	VAR robtarget Openhole_2763 := [[394.33, -31.54, 174.56], [-0.132881, 0.694509, 0.676037, 0.207303], [0,0,0,0], [9E9, 9E9, 9E9, 9E9, 9E9, 9E9]];
	VAR robtarget Openhole_2764 := [[389.32, -31.54, 173.95], [-0.146442, 0.691776, 0.672345, 0.218979], [0,0,0,0], [9E9, 9E9, 9E9, 9E9, 9E9, 9E9]];
	VAR robtarget Openhole_2765 := [[362.32, -31.54, 174.04], [-0.183051, 0.683002, 0.683002, 0.183051], [0,0,0,0], [9E9, 9E9, 9E9, 9E9, 9E9, 9E9]];
	VAR robtarget Openhole_2766 := [[362.32, -32.55, 173.46], [-0.183051, 0.683002, 0.683002, 0.183051], [0,0,0,0], [9E9, 9E9, 9E9, 9E9, 9E9, 9E9]];
	VAR robtarget Openhole_2767 := [[389.32, -32.55, 173.37], [-0.143577, 0.692377, 0.671432, 0.221765], [0,0,0,0], [9E9, 9E9, 9E9, 9E9, 9E9, 9E9]];
	VAR robtarget Openhole_2768 := [[394.32, -32.55, 174.02], [-0.129957, 0.695062, 0.675151, 0.210168], [0,0,0,0], [9E9, 9E9, 9E9, 9E9, 9E9, 9E9]];
	VAR robtarget Openhole_2769 := [[395.25, -32.64, 174.1], [-0.127122, 0.695586, 0.675755, 0.20822], [0,0,0,0], [9E9, 9E9, 9E9, 9E9, 9E9, 9E9]];
	VAR robtarget Openhole_2770 := [[405.09, -34.29, 174.68], [-0.093512, 0.700896, 0.681563, 0.188339], [0,0,0,0], [9E9, 9E9, 9E9, 9E9, 9E9, 9E9]];
	VAR robtarget Openhole_2771 := [[411.51, -35.11, 175.33], [-0.071164, 0.703517, 0.685468, 0.173589], [0,0,0,0], [9E9, 9E9, 9E9, 9E9, 9E9, 9E9]];
	VAR robtarget Openhole_2772 := [[417.44, -35.57, 176.1], [-0.050738, 0.705284, 0.689168, 0.158265], [0,0,0,0], [9E9, 9E9, 9E9, 9E9, 9E9, 9E9]];
	VAR robtarget Openhole_2773 := [[421.88, -35.68, 176.78], [-0.035801, 0.7062, 0.691962, 0.145564], [0,0,0,0], [9E9, 9E9, 9E9, 9E9, 9E9, 9E9]];
	VAR robtarget Openhole_2774 := [[422.38, -35.68, 176.86], [-0.034176, 0.70628, 0.692272, 0.14408], [0,0,0,0], [9E9, 9E9, 9E9, 9E9, 9E9, 9E9]];
	VAR robtarget Openhole_2775 := [[428.29, -35.44, 177.86], [-0.015185, 0.706944, 0.695923, 0.125263], [0,0,0,0], [9E9, 9E9, 9E9, 9E9, 9E9, 9E9]];
	VAR robtarget Openhole_2776 := [[436.16, -34.91, 179.17], [0.00982, 0.707039, 0.700215, 0.098481], [0,0,0,0], [9E9, 9E9, 9E9, 9E9, 9E9, 9E9]];
	VAR robtarget Openhole_2777 := [[437.15, -34.9, 179.32], [0.013143, 0.706985, 0.700667, 0.095213], [0,0,0,0], [9E9, 9E9, 9E9, 9E9, 9E9, 9E9]];
	VAR robtarget Openhole_2778 := [[437.64, -34.9, 179.39], [0.014832, 0.706951, 0.700885, 0.093599], [0,0,0,0], [9E9, 9E9, 9E9, 9E9, 9E9, 9E9]];
	VAR robtarget Openhole_2779 := [[439.13, -34.94, 179.62], [0.020035, 0.706823, 0.7015, 0.088866], [0,0,0,0], [9E9, 9E9, 9E9, 9E9, 9E9, 9E9]];
	VAR robtarget Openhole_2780 := [[440.11, -35, 179.76], [0.023624, 0.706712, 0.701879, 0.085823], [0,0,0,0], [9E9, 9E9, 9E9, 9E9, 9E9, 9E9]];
	VAR robtarget Openhole_2781 := [[443.54, -35.46, 180.26], [0.036875, 0.706145, 0.703018, 0.075935], [0,0,0,0], [9E9, 9E9, 9E9, 9E9, 9E9, 9E9]];
	VAR robtarget Openhole_2782 := [[446.93, -36.18, 180.78], [0.05077, 0.705282, 0.703935, 0.066903], [0,0,0,0], [9E9, 9E9, 9E9, 9E9, 9E9, 9E9]];
	VAR robtarget Openhole_2783 := [[447.42, -36.26, 180.86], [0.052703, 0.70514, 0.704063, 0.065541], [0,0,0,0], [9E9, 9E9, 9E9, 9E9, 9E9, 9E9]];
	VAR robtarget Openhole_2784 := [[447.91, -36.33, 180.94], [0.054605, 0.704995, 0.704192, 0.064136], [0,0,0,0], [9E9, 9E9, 9E9, 9E9, 9E9, 9E9]];
	VAR robtarget Openhole_2785 := [[448.4, -36.38, 181.02], [0.056429, 0.704852, 0.704327, 0.062633], [0,0,0,0], [9E9, 9E9, 9E9, 9E9, 9E9, 9E9]];
	VAR robtarget Openhole_2786 := [[448.89, -36.4, 181.11], [0.058152, 0.704712, 0.70447, 0.061014], [0,0,0,0], [9E9, 9E9, 9E9, 9E9, 9E9, 9E9]];
	VAR robtarget Openhole_2787 := [[449.38, -36.38, 181.19], [0.059774, 0.704576, 0.704616, 0.059293], [0,0,0,0], [9E9, 9E9, 9E9, 9E9, 9E9, 9E9]];
	VAR robtarget Openhole_2788 := [[449.87, -36.33, 181.27], [0.061269, 0.704447, 0.704768, 0.057463], [0,0,0,0], [9E9, 9E9, 9E9, 9E9, 9E9, 9E9]];
	VAR robtarget Openhole_2789 := [[450.85, -36.17, 181.43], [0.064011, 0.704203, 0.705072, 0.053608], [0,0,0,0], [9E9, 9E9, 9E9, 9E9, 9E9, 9E9]];
	VAR robtarget Openhole_2790 := [[455.16, -35.07, 182.08], [0.074877, 0.703131, 0.706227, 0.035254], [0,0,0,0], [9E9, 9E9, 9E9, 9E9, 9E9, 9E9]];
	VAR robtarget Openhole_2791 := [[460.92, -33.54, 182.8], [0.08889, 0.701497, 0.707029, 0.010492], [0,0,0,0], [9E9, 9E9, 9E9, 9E9, 9E9, 9E9]];
	VAR robtarget Openhole_2792 := [[466.77, -32.38, 183.42], [0.104054, 0.699409, 0.706982, -0.013257], [0,0,0,0], [9E9, 9E9, 9E9, 9E9, 9E9, 9E9]];
	VAR robtarget Openhole_2793 := [[473.67, -31.4, 184.08], [0.122541, 0.696408, 0.705996, -0.039613], [0,0,0,0], [9E9, 9E9, 9E9, 9E9, 9E9, 9E9]];
	VAR robtarget Openhole_2794 := [[482.09, -30.56, 184.82], [0.145189, 0.692041, 0.703659, -0.069743], [0,0,0,0], [9E9, 9E9, 9E9, 9E9, 9E9, 9E9]];
	VAR robtarget Openhole_2795 := [[494.53, -29.79, 185.86], [0.177448, 0.68448, 0.698437, -0.110387], [0,0,0,0], [9E9, 9E9, 9E9, 9E9, 9E9, 9E9]];
	VAR robtarget Openhole_2796 := [[504.36, -29.28, 186.61], [0.200859, 0.677979, 0.693127, -0.13991], [0,0,0,0], [9E9, 9E9, 9E9, 9E9, 9E9, 9E9]];
	VAR robtarget Openhole_2797 := [[509.36, -29.28, 187.1], [0.183051, 0.683002, 0.683002, -0.183051], [0,0,0,0], [9E9, 9E9, 9E9, 9E9, 9E9, 9E9]];
	VAR robtarget Openhole_2798 := [[536.36, -29.28, 187.02], [0.183051, 0.683002, 0.683002, -0.183051], [0,0,0,0], [9E9, 9E9, 9E9, 9E9, 9E9, 9E9]];
	VAR robtarget Openhole_2799 := [[536.37, -30.16, 187.53], [0.183051, 0.683002, 0.683002, -0.183051], [0,0,0,0], [9E9, 9E9, 9E9, 9E9, 9E9, 9E9]];
	VAR robtarget Openhole_2800 := [[524.37, -30.16, 187.56], [0.183051, 0.683002, 0.683002, -0.183051], [0,0,0,0], [9E9, 9E9, 9E9, 9E9, 9E9, 9E9]];
	VAR robtarget Openhole_2801 := [[509.37, -30.16, 187.61], [0.183051, 0.683002, 0.683002, -0.183051], [0,0,0,0], [9E9, 9E9, 9E9, 9E9, 9E9, 9E9]];
	VAR robtarget Openhole_2802 := [[504.38, -30.16, 187.08], [0.203409, 0.677218, 0.693637, -0.13736], [0,0,0,0], [9E9, 9E9, 9E9, 9E9, 9E9, 9E9]];
	VAR robtarget Openhole_2803 := [[485.97, -31.27, 185.5], [0.158522, 0.689109, 0.702598, -0.079726], [0,0,0,0], [9E9, 9E9, 9E9, 9E9, 9E9, 9E9]];
	VAR robtarget Openhole_2804 := [[477.54, -32.07, 184.72], [0.136459, 0.693815, 0.705324, -0.050181], [0,0,0,0], [9E9, 9E9, 9E9, 9E9, 9E9, 9E9]];
	VAR robtarget Openhole_2805 := [[470.15, -33.11, 184], [0.117126, 0.697339, 0.706757, -0.022242], [0,0,0,0], [9E9, 9E9, 9E9, 9E9, 9E9, 9E9]];
	VAR robtarget Openhole_2806 := [[463.32, -34.47, 183.26], [0.099767, 0.700033, 0.707086, 0.005357], [0,0,0,0], [9E9, 9E9, 9E9, 9E9, 9E9, 9E9]];
	VAR robtarget Openhole_2807 := [[457.09, -36.14, 182.46], [0.084833, 0.702, 0.706374, 0.032194], [0,0,0,0], [9E9, 9E9, 9E9, 9E9, 9E9, 9E9]];
	VAR robtarget Openhole_2808 := [[450.91, -37.89, 181.47], [0.069901, 0.703643, 0.704636, 0.059065], [0,0,0,0], [9E9, 9E9, 9E9, 9E9, 9E9, 9E9]];
	VAR robtarget Openhole_2809 := [[449.96, -38.12, 181.29], [0.067407, 0.703887, 0.704289, 0.063064], [0,0,0,0], [9E9, 9E9, 9E9, 9E9, 9E9, 9E9]];
	VAR robtarget Openhole_2810 := [[449.47, -38.19, 181.2], [0.065977, 0.704022, 0.704119, 0.064933], [0,0,0,0], [9E9, 9E9, 9E9, 9E9, 9E9, 9E9]];
	VAR robtarget Openhole_2811 := [[448.98, -38.23, 181.11], [0.064462, 0.704162, 0.70395, 0.066738], [0,0,0,0], [9E9, 9E9, 9E9, 9E9, 9E9, 9E9]];
	VAR robtarget Openhole_2812 := [[448.49, -38.23, 181.02], [0.062791, 0.704313, 0.703791, 0.068398], [0,0,0,0], [9E9, 9E9, 9E9, 9E9, 9E9, 9E9]];
	VAR robtarget Openhole_2813 := [[448, -38.2, 180.93], [0.061046, 0.704467, 0.703636, 0.069978], [0,0,0,0], [9E9, 9E9, 9E9, 9E9, 9E9, 9E9]];
	VAR robtarget Openhole_2814 := [[447.51, -38.14, 180.84], [0.05919, 0.704625, 0.70349, 0.071428], [0,0,0,0], [9E9, 9E9, 9E9, 9E9, 9E9, 9E9]];
	VAR robtarget Openhole_2815 := [[447.02, -38.07, 180.76], [0.057282, 0.704783, 0.703348, 0.072811], [0,0,0,0], [9E9, 9E9, 9E9, 9E9, 9E9, 9E9]];
	VAR robtarget Openhole_2816 := [[446.06, -37.84, 180.59], [0.053281, 0.705097, 0.703085, 0.075305], [0,0,0,0], [9E9, 9E9, 9E9, 9E9, 9E9, 9E9]];
	VAR robtarget Openhole_2817 := [[445.11, -37.59, 180.42], [0.049204, 0.705393, 0.702827, 0.077681], [0,0,0,0], [9E9, 9E9, 9E9, 9E9, 9E9, 9E9]];
	VAR robtarget Openhole_2818 := [[444.14, -37.38, 180.26], [0.045235, 0.705658, 0.70254, 0.080239], [0,0,0,0], [9E9, 9E9, 9E9, 9E9, 9E9, 9E9]];
	VAR robtarget Openhole_2819 := [[443.17, -37.22, 180.1], [0.04138, 0.705895, 0.702223, 0.08296], [0,0,0,0], [9E9, 9E9, 9E9, 9E9, 9E9, 9E9]];
	VAR robtarget Openhole_2820 := [[442.19, -37.1, 179.94], [0.037628, 0.706105, 0.701881, 0.085812], [0,0,0,0], [9E9, 9E9, 9E9, 9E9, 9E9, 9E9]];
	VAR robtarget Openhole_2821 := [[438.25, -36.86, 179.28], [0.023389, 0.70672, 0.700279, 0.098025], [0,0,0,0], [9E9, 9E9, 9E9, 9E9, 9E9, 9E9]];
	VAR robtarget Openhole_2822 := [[437.76, -36.86, 179.19], [0.021703, 0.706774, 0.700052, 0.099635], [0,0,0,0], [9E9, 9E9, 9E9, 9E9, 9E9, 9E9]];
	VAR robtarget Openhole_2823 := [[437.27, -36.86, 179.11], [0.020021, 0.706823, 0.699821, 0.101245], [0,0,0,0], [9E9, 9E9, 9E9, 9E9, 9E9, 9E9]];
	VAR robtarget Openhole_2824 := [[429.9, -37.22, 177.78], [-0.003966, 0.707096, 0.695802, 0.125933], [0,0,0,0], [9E9, 9E9, 9E9, 9E9, 9E9, 9E9]];
	VAR robtarget Openhole_2825 := [[424, -37.4, 176.7], [-0.023235, 0.706725, 0.692154, 0.144649], [0,0,0,0], [9E9, 9E9, 9E9, 9E9, 9E9, 9E9]];
	VAR robtarget Openhole_2826 := [[423.5, -37.4, 176.61], [-0.02488, 0.706669, 0.691843, 0.146127], [0,0,0,0], [9E9, 9E9, 9E9, 9E9, 9E9, 9E9]];
	VAR robtarget Openhole_2827 := [[417.59, -37.22, 175.62], [-0.045011, 0.705673, 0.688083, 0.162916], [0,0,0,0], [9E9, 9E9, 9E9, 9E9, 9E9, 9E9]];
	VAR robtarget Openhole_2828 := [[411.67, -36.7, 174.78], [-0.065682, 0.70405, 0.684353, 0.177935], [0,0,0,0], [9E9, 9E9, 9E9, 9E9, 9E9, 9E9]];
	VAR robtarget Openhole_2829 := [[405.77, -35.88, 174.12], [-0.086593, 0.701785, 0.680742, 0.191285], [0,0,0,0], [9E9, 9E9, 9E9, 9E9, 9E9, 9E9]];
	VAR robtarget Openhole_2830 := [[399.88, -34.8, 173.68], [-0.107456, 0.698894, 0.677313, 0.203095], [0,0,0,0], [9E9, 9E9, 9E9, 9E9, 9E9, 9E9]];
	VAR robtarget Openhole_2831 := [[395, -33.77, 173.47], [-0.124525, 0.696056, 0.674576, 0.212008], [0,0,0,0], [9E9, 9E9, 9E9, 9E9, 9E9, 9E9]];
	VAR robtarget Openhole_2832 := [[394.32, -33.65, 173.44], [-0.126742, 0.695655, 0.674171, 0.213293], [0,0,0,0], [9E9, 9E9, 9E9, 9E9, 9E9, 9E9]];
	VAR robtarget Openhole_2833 := [[389.32, -33.65, 172.73], [-0.140438, 0.69302, 0.670418, 0.224811], [0,0,0,0], [9E9, 9E9, 9E9, 9E9, 9E9, 9E9]];
	VAR robtarget Openhole_2834 := [[362.32, -33.65, 172.82], [-0.183051, 0.683002, 0.683002, 0.183051], [0,0,0,0], [9E9, 9E9, 9E9, 9E9, 9E9, 9E9]];
	VAR robtarget Openhole_2835 := [[362.32, -34.53, 172.31], [-0.183051, 0.683002, 0.683002, 0.183051], [0,0,0,0], [9E9, 9E9, 9E9, 9E9, 9E9, 9E9]];
	VAR robtarget Openhole_2836 := [[374.32, -34.53, 172.27], [-0.183051, 0.683002, 0.683002, 0.183051], [0,0,0,0], [9E9, 9E9, 9E9, 9E9, 9E9, 9E9]];
	VAR robtarget Openhole_2837 := [[389.32, -34.53, 172.23], [-0.137959, 0.693518, 0.669608, 0.227211], [0,0,0,0], [9E9, 9E9, 9E9, 9E9, 9E9, 9E9]];
	VAR robtarget Openhole_2838 := [[394.23, -34.53, 172.96], [-0.124447, 0.69607, 0.673324, 0.21595], [0,0,0,0], [9E9, 9E9, 9E9, 9E9, 9E9, 9E9]];
	VAR robtarget Openhole_2839 := [[400.62, -36.11, 173.18], [-0.101392, 0.6998, 0.676729, 0.205033], [0,0,0,0], [9E9, 9E9, 9E9, 9E9, 9E9, 9E9]];
	VAR robtarget Openhole_2840 := [[406, -37.14, 173.63], [-0.082029, 0.702333, 0.67986, 0.194398], [0,0,0,0], [9E9, 9E9, 9E9, 9E9, 9E9, 9E9]];
	VAR robtarget Openhole_2841 := [[412.39, -38.07, 174.41], [-0.059148, 0.704629, 0.68378, 0.180126], [0,0,0,0], [9E9, 9E9, 9E9, 9E9, 9E9, 9E9]];
	VAR robtarget Openhole_2842 := [[418.29, -38.63, 175.33], [-0.038284, 0.70607, 0.68753, 0.165233], [0,0,0,0], [9E9, 9E9, 9E9, 9E9, 9E9, 9E9]];
	VAR robtarget Openhole_2843 := [[418.78, -38.66, 175.41], [-0.036565, 0.706161, 0.687846, 0.163914], [0,0,0,0], [9E9, 9E9, 9E9, 9E9, 9E9, 9E9]];
	VAR robtarget Openhole_2844 := [[419.27, -38.7, 175.49], [-0.034805, 0.70625, 0.688152, 0.162624], [0,0,0,0], [9E9, 9E9, 9E9, 9E9, 9E9, 9E9]];
	VAR robtarget Openhole_2845 := [[408.81, -38.7, 173.51], [-0.068565, 0.703775, 0.680645, 0.191632], [0,0,0,0], [9E9, 9E9, 9E9, 9E9, 9E9, 9E9]];
	VAR robtarget Openhole_2846 := [[408.32, -38.6, 173.46], [-0.070405, 0.703593, 0.680359, 0.192643], [0,0,0,0], [9E9, 9E9, 9E9, 9E9, 9E9, 9E9]];
	VAR robtarget Openhole_2847 := [[402.93, -37.64, 172.87], [-0.089888, 0.70137, 0.677133, 0.203693], [0,0,0,0], [9E9, 9E9, 9E9, 9E9, 9E9, 9E9]];
	VAR robtarget Openhole_2848 := [[398.07, -36.52, 172.56], [-0.107652, 0.698864, 0.674439, 0.212442], [0,0,0,0], [9E9, 9E9, 9E9, 9E9, 9E9, 9E9]];
	VAR robtarget Openhole_2849 := [[395.19, -35.69, 172.5], [-0.118358, 0.697131, 0.672991, 0.216986], [0,0,0,0], [9E9, 9E9, 9E9, 9E9, 9E9, 9E9]];
	VAR robtarget Openhole_2850 := [[394.71, -35.54, 172.5], [-0.120156, 0.696823, 0.672771, 0.217667], [0,0,0,0], [9E9, 9E9, 9E9, 9E9, 9E9, 9E9]];
	VAR robtarget Openhole_2851 := [[394.32, -35.51, 172.46], [-0.121349, 0.696616, 0.672496, 0.218517], [0,0,0,0], [9E9, 9E9, 9E9, 9E9, 9E9, 9E9]];
	VAR robtarget Openhole_2852 := [[389.32, -35.51, 171.66], [-0.13517, 0.694067, 0.668688, 0.229905], [0,0,0,0], [9E9, 9E9, 9E9, 9E9, 9E9, 9E9]];
	VAR robtarget Openhole_2853 := [[360.24, -35.51, 171.75], [-0.183051, 0.683002, 0.683002, 0.183051], [0,0,0,0], [9E9, 9E9, 9E9, 9E9, 9E9, 9E9]];
	VAR robtarget Openhole_2854 := [[360.28, -11.45, 185.65], [-0.183051, 0.683002, 0.683002, 0.183051], [0,0,0,0], [9E9, 9E9, 9E9, 9E9, 9E9, 9E9]];
	VAR robtarget Openhole_2855 := [[389.36, -11.45, 185.56], [-0.203596, 0.677162, 0.688281, 0.162077], [0,0,0,0], [9E9, 9E9, 9E9, 9E9, 9E9, 9E9]];
	VAR robtarget Openhole_2856 := [[394.36, -11.45, 185.19], [-0.191483, 0.680686, 0.691238, 0.148963], [0,0,0,0], [9E9, 9E9, 9E9, 9E9, 9E9, 9E9]];
	VAR robtarget Openhole_2857 := [[406.15, -10.95, 184.54], [-0.162117, 0.688272, 0.697809, 0.114295], [0,0,0,0], [9E9, 9E9, 9E9, 9E9, 9E9, 9E9]];
	VAR robtarget Openhole_2858 := [[427.08, -10.18, 183.08], [-0.102415, 0.699651, 0.7056, 0.046144], [0,0,0,0], [9E9, 9E9, 9E9, 9E9, 9E9, 9E9]];
	VAR robtarget Openhole_2859 := [[441.52, -9.59, 181.89], [-0.057181, 0.704791, 0.707093, -0.004439], [0,0,0,0], [9E9, 9E9, 9E9, 9E9, 9E9, 9E9]];
	VAR robtarget Openhole_2860 := [[443.51, -9.49, 181.72], [-0.050801, 0.70528, 0.707013, -0.01153], [0,0,0,0], [9E9, 9E9, 9E9, 9E9, 9E9, 9E9]];
	VAR robtarget Openhole_2861 := [[445.01, -9.52, 181.58], [-0.045692, 0.705629, 0.706913, -0.016552], [0,0,0,0], [9E9, 9E9, 9E9, 9E9, 9E9, 9E9]];
	VAR robtarget Openhole_2862 := [[447, -9.62, 181.39], [-0.038623, 0.706051, 0.706733, -0.022994], [0,0,0,0], [9E9, 9E9, 9E9, 9E9, 9E9, 9E9]];
	VAR robtarget Openhole_2863 := [[450.48, -9.77, 181.08], [-0.026284, 0.706618, 0.706273, -0.034334], [0,0,0,0], [9E9, 9E9, 9E9, 9E9, 9E9, 9E9]];
	VAR robtarget Openhole_2864 := [[451.47, -9.76, 180.99], [-0.022937, 0.706735, 0.706098, -0.037759], [0,0,0,0], [9E9, 9E9, 9E9, 9E9, 9E9, 9E9]];
	VAR robtarget Openhole_2865 := [[452.96, -9.66, 180.86], [-0.018189, 0.706873, 0.70579, -0.043139], [0,0,0,0], [9E9, 9E9, 9E9, 9E9, 9E9, 9E9]];
	VAR robtarget Openhole_2866 := [[453.46, -9.61, 180.81], [-0.016656, 0.706911, 0.705675, -0.044972], [0,0,0,0], [9E9, 9E9, 9E9, 9E9, 9E9, 9E9]];
	VAR robtarget Openhole_2867 := [[453.95, -9.56, 180.76], [-0.015166, 0.706944, 0.705554, -0.046838], [0,0,0,0], [9E9, 9E9, 9E9, 9E9, 9E9, 9E9]];
	VAR robtarget Openhole_2868 := [[456.91, -9.15, 180.46], [-0.006451, 0.707077, 0.704711, -0.058155], [0,0,0,0], [9E9, 9E9, 9E9, 9E9, 9E9, 9E9]];
	VAR robtarget Openhole_2869 := [[464.72, -7.68, 179.5], [0.015109, 0.706945, 0.701497, -0.088892], [0,0,0,0], [9E9, 9E9, 9E9, 9E9, 9E9, 9E9]];
	VAR robtarget Openhole_2870 := [[471.06, -6.59, 178.58], [0.032782, 0.706346, 0.698055, -0.112783], [0,0,0,0], [9E9, 9E9, 9E9, 9E9, 9E9, 9E9]];
	VAR robtarget Openhole_2871 := [[475.49, -6.13, 177.94], [0.045922, 0.705614, 0.695421, -0.128021], [0,0,0,0], [9E9, 9E9, 9E9, 9E9, 9E9, 9E9]];
	VAR robtarget Openhole_2872 := [[479.94, -5.98, 177.34], [0.059908, 0.704564, 0.692711, -0.141955], [0,0,0,0], [9E9, 9E9, 9E9, 9E9, 9E9, 9E9]];
	VAR robtarget Openhole_2873 := [[480.44, -5.98, 177.28], [0.061506, 0.704427, 0.692408, -0.143424], [0,0,0,0], [9E9, 9E9, 9E9, 9E9, 9E9, 9E9]];
	VAR robtarget Openhole_2874 := [[485.9, -6.15, 176.65], [0.079354, 0.70264, 0.689063, -0.158719], [0,0,0,0], [9E9, 9E9, 9E9, 9E9, 9E9, 9E9]];
	VAR robtarget Openhole_2875 := [[495.33, -6.89, 175.81], [0.110212, 0.698465, 0.68321, -0.182276], [0,0,0,0], [9E9, 9E9, 9E9, 9E9, 9E9, 9E9]];
	VAR robtarget Openhole_2876 := [[501.3, -7.34, 175.33], [0.128643, 0.695306, 0.67933, -0.19624], [0,0,0,0], [9E9, 9E9, 9E9, 9E9, 9E9, 9E9]];
	VAR robtarget Openhole_2877 := [[504.33, -7.39, 175.02], [0.137193, 0.69367, 0.677182, -0.20353], [0,0,0,0], [9E9, 9E9, 9E9, 9E9, 9E9, 9E9]];
	VAR robtarget Openhole_2878 := [[509.32, -7.39, 174.46], [0.183051, 0.683002, 0.683002, -0.183051], [0,0,0,0], [9E9, 9E9, 9E9, 9E9, 9E9, 9E9]];
	VAR robtarget Openhole_2879 := [[536.32, -7.39, 174.38], [0.183051, 0.683002, 0.683002, -0.183051], [0,0,0,0], [9E9, 9E9, 9E9, 9E9, 9E9, 9E9]];
	VAR robtarget Openhole_2880 := [[536.32, -6.51, 173.87], [0.183051, 0.683002, 0.683002, -0.183051], [0,0,0,0], [9E9, 9E9, 9E9, 9E9, 9E9, 9E9]];
	VAR robtarget Openhole_2881 := [[509.32, -6.51, 173.95], [0.183051, 0.683002, 0.683002, -0.183051], [0,0,0,0], [9E9, 9E9, 9E9, 9E9, 9E9, 9E9]];
	VAR robtarget Openhole_2882 := [[504.33, -6.51, 174.55], [0.134614, 0.694175, 0.676421, -0.206046], [0,0,0,0], [9E9, 9E9, 9E9, 9E9, 9E9, 9E9]];
	VAR robtarget Openhole_2883 := [[504.3, -6.51, 174.56], [0.134528, 0.694192, 0.676442, -0.205978], [0,0,0,0], [9E9, 9E9, 9E9, 9E9, 9E9, 9E9]];
	VAR robtarget Openhole_2884 := [[503.8, -6.51, 174.62], [0.133159, 0.694456, 0.676805, -0.20478], [0,0,0,0], [9E9, 9E9, 9E9, 9E9, 9E9, 9E9]];
	VAR robtarget Openhole_2885 := [[498.83, -6.2, 175.07], [0.118278, 0.697144, 0.680159, -0.19335], [0,0,0,0], [9E9, 9E9, 9E9, 9E9, 9E9, 9E9]];
	VAR robtarget Openhole_2886 := [[488.43, -5.09, 175.94], [0.083887, 0.702113, 0.6866, -0.169059], [0,0,0,0], [9E9, 9E9, 9E9, 9E9, 9E9, 9E9]];
	VAR robtarget Openhole_2887 := [[481.98, -4.67, 176.67], [0.062284, 0.704358, 0.690563, -0.152061], [0,0,0,0], [9E9, 9E9, 9E9, 9E9, 9E9, 9E9]];
	VAR robtarget Openhole_2888 := [[478.51, -4.61, 177.13], [0.0509, 0.705272, 0.692697, -0.142022], [0,0,0,0], [9E9, 9E9, 9E9, 9E9, 9E9, 9E9]];
	VAR robtarget Openhole_2889 := [[478.02, -4.61, 177.2], [0.0493, 0.705386, 0.693002, -0.14053], [0,0,0,0], [9E9, 9E9, 9E9, 9E9, 9E9, 9E9]];
	VAR robtarget Openhole_2890 := [[473.08, -4.83, 177.94], [0.033725, 0.706302, 0.696006, -0.124805], [0,0,0,0], [9E9, 9E9, 9E9, 9E9, 9E9, 9E9]];
	VAR robtarget Openhole_2891 := [[466.69, -5.54, 178.93], [0.014683, 0.706954, 0.699661, -0.102346], [0,0,0,0], [9E9, 9E9, 9E9, 9E9, 9E9, 9E9]];
	VAR robtarget Openhole_2892 := [[463.75, -5.92, 179.36], [0.005993, 0.707081, 0.701154, -0.091561], [0,0,0,0], [9E9, 9E9, 9E9, 9E9, 9E9, 9E9]];
	VAR robtarget Openhole_2893 := [[461.29, -6.17, 179.7], [-0.001528, 0.707105, 0.702261, -0.082644], [0,0,0,0], [9E9, 9E9, 9E9, 9E9, 9E9, 9E9]];
	VAR robtarget Openhole_2894 := [[460.3, -6.24, 179.83], [-0.004665, 0.707091, 0.702663, -0.079151], [0,0,0,0], [9E9, 9E9, 9E9, 9E9, 9E9, 9E9]];
	VAR robtarget Openhole_2895 := [[459.31, -6.28, 179.96], [-0.0079, 0.707063, 0.70304, -0.075728], [0,0,0,0], [9E9, 9E9, 9E9, 9E9, 9E9, 9E9]];
	VAR robtarget Openhole_2896 := [[458.31, -6.3, 180.08], [-0.01123, 0.707018, 0.703393, -0.072376], [0,0,0,0], [9E9, 9E9, 9E9, 9E9, 9E9, 9E9]];
	VAR robtarget Openhole_2897 := [[457.82, -6.3, 180.14], [-0.012928, 0.706989, 0.703561, -0.070727], [0,0,0,0], [9E9, 9E9, 9E9, 9E9, 9E9, 9E9]];
	VAR robtarget Openhole_2898 := [[457.32, -6.28, 180.2], [-0.014668, 0.706955, 0.70372, -0.06912], [0,0,0,0], [9E9, 9E9, 9E9, 9E9, 9E9, 9E9]];
	VAR robtarget Openhole_2899 := [[452.38, -5.84, 180.8], [-0.033015, 0.706336, 0.705043, -0.053983], [0,0,0,0], [9E9, 9E9, 9E9, 9E9, 9E9, 9E9]];
	VAR robtarget Openhole_2900 := [[450.4, -5.64, 181.04], [-0.040416, 0.705951, 0.705477, -0.047977], [0,0,0,0], [9E9, 9E9, 9E9, 9E9, 9E9, 9E9]];
	VAR robtarget Openhole_2901 := [[448.92, -5.55, 181.24], [-0.045754, 0.705625, 0.705784, -0.043224], [0,0,0,0], [9E9, 9E9, 9E9, 9E9, 9E9, 9E9]];
	VAR robtarget Openhole_2902 := [[448.42, -5.54, 181.3], [-0.047464, 0.705512, 0.705884, -0.041566], [0,0,0,0], [9E9, 9E9, 9E9, 9E9, 9E9, 9E9]];
	VAR robtarget Openhole_2903 := [[447.93, -5.54, 181.37], [-0.049134, 0.705398, 0.705982, -0.039867], [0,0,0,0], [9E9, 9E9, 9E9, 9E9, 9E9, 9E9]];
	VAR robtarget Openhole_2904 := [[447.43, -5.56, 181.43], [-0.050738, 0.705284, 0.706079, -0.038106], [0,0,0,0], [9E9, 9E9, 9E9, 9E9, 9E9, 9E9]];
	VAR robtarget Openhole_2905 := [[446.94, -5.6, 181.49], [-0.052288, 0.705171, 0.706175, -0.036296], [0,0,0,0], [9E9, 9E9, 9E9, 9E9, 9E9, 9E9]];
	VAR robtarget Openhole_2906 := [[446.44, -5.65, 181.56], [-0.053794, 0.705058, 0.706267, -0.034449], [0,0,0,0], [9E9, 9E9, 9E9, 9E9, 9E9, 9E9]];
	VAR robtarget Openhole_2907 := [[445.46, -5.78, 181.68], [-0.056696, 0.70483, 0.706441, -0.030668], [0,0,0,0], [9E9, 9E9, 9E9, 9E9, 9E9, 9E9]];
	VAR robtarget Openhole_2908 := [[437.62, -7.11, 182.53], [-0.078428, 0.702744, 0.707107, 0.000556], [0,0,0,0], [9E9, 9E9, 9E9, 9E9, 9E9, 9E9]];
	VAR robtarget Openhole_2909 := [[429.7, -8.01, 183.27], [-0.101196, 0.699828, 0.706459, 0.03026], [0,0,0,0], [9E9, 9E9, 9E9, 9E9, 9E9, 9E9]];
	VAR robtarget Openhole_2910 := [[418.28, -8.88, 184.22], [-0.133751, 0.694342, 0.703582, 0.070513], [0,0,0,0], [9E9, 9E9, 9E9, 9E9, 9E9, 9E9]];
	VAR robtarget Openhole_2911 := [[396.86, -9.88, 185.8], [-0.189787, 0.681161, 0.693603, 0.13753], [0,0,0,0], [9E9, 9E9, 9E9, 9E9, 9E9, 9E9]];
	VAR robtarget Openhole_2912 := [[394.36, -10.02, 185.95], [-0.195594, 0.679517, 0.692127, 0.144776], [0,0,0,0], [9E9, 9E9, 9E9, 9E9, 9E9, 9E9]];
	VAR robtarget Openhole_2913 := [[389.36, -10.02, 186.38], [-0.207603, 0.675944, 0.689231, 0.157991], [0,0,0,0], [9E9, 9E9, 9E9, 9E9, 9E9, 9E9]];
	VAR robtarget Openhole_2914 := [[362.36, -10.02, 186.47], [-0.183051, 0.683002, 0.683002, 0.183051], [0,0,0,0], [9E9, 9E9, 9E9, 9E9, 9E9, 9E9]];
	VAR robtarget Openhole_2915 := [[362.36, -9.02, 187.04], [-0.183051, 0.683002, 0.683002, 0.183051], [0,0,0,0], [9E9, 9E9, 9E9, 9E9, 9E9, 9E9]];
	VAR robtarget Openhole_2916 := [[389.36, -9.02, 186.96], [-0.210402, 0.675079, 0.68988, 0.15513], [0,0,0,0], [9E9, 9E9, 9E9, 9E9, 9E9, 9E9]];
	VAR robtarget Openhole_2917 := [[394.36, -9.02, 186.48], [-0.198465, 0.678684, 0.692734, 0.141845], [0,0,0,0], [9E9, 9E9, 9E9, 9E9, 9E9, 9E9]];
	VAR robtarget Openhole_2918 := [[414.68, -7.96, 184.87], [-0.14724, 0.691607, 0.702683, 0.078975], [0,0,0,0], [9E9, 9E9, 9E9, 9E9, 9E9, 9E9]];
	VAR robtarget Openhole_2919 := [[424.61, -7.15, 184.01], [-0.120013, 0.696848, 0.705713, 0.044371], [0,0,0,0], [9E9, 9E9, 9E9, 9E9, 9E9, 9E9]];
	VAR robtarget Openhole_2920 := [[432.02, -6.25, 183.31], [-0.09953, 0.700067, 0.70691, 0.016666], [0,0,0,0], [9E9, 9E9, 9E9, 9E9, 9E9, 9E9]];
	VAR robtarget Openhole_2921 := [[438.39, -5.14, 182.65], [-0.082413, 0.702288, 0.707054, -0.008641], [0,0,0,0], [9E9, 9E9, 9E9, 9E9, 9E9, 9E9]];
	VAR robtarget Openhole_2922 := [[446.11, -3.31, 181.67], [-0.0627, 0.704321, 0.705909, -0.041135], [0,0,0,0], [9E9, 9E9, 9E9, 9E9, 9E9, 9E9]];
	VAR robtarget Openhole_2923 := [[447.09, -3.15, 181.53], [-0.059927, 0.704563, 0.705674, -0.044991], [0,0,0,0], [9E9, 9E9, 9E9, 9E9, 9E9, 9E9]];
	VAR robtarget Openhole_2924 := [[447.58, -3.09, 181.45], [-0.058485, 0.704684, 0.705551, -0.046877], [0,0,0,0], [9E9, 9E9, 9E9, 9E9, 9E9, 9E9]];
	VAR robtarget Openhole_2925 := [[448.07, -3.04, 181.38], [-0.056976, 0.704808, 0.705427, -0.04871], [0,0,0,0], [9E9, 9E9, 9E9, 9E9, 9E9, 9E9]];
	VAR robtarget Openhole_2926 := [[448.57, -3, 181.3], [-0.055435, 0.70493, 0.7053, -0.050514], [0,0,0,0], [9E9, 9E9, 9E9, 9E9, 9E9, 9E9]];
	VAR robtarget Openhole_2927 := [[449.06, -3, 181.23], [-0.053771, 0.705059, 0.705177, -0.052205], [0,0,0,0], [9E9, 9E9, 9E9, 9E9, 9E9, 9E9]];
	VAR robtarget Openhole_2928 := [[449.55, -3.01, 181.15], [-0.052051, 0.705188, 0.705054, -0.05384], [0,0,0,0], [9E9, 9E9, 9E9, 9E9, 9E9, 9E9]];
	VAR robtarget Openhole_2929 := [[450.54, -3.1, 181], [-0.048406, 0.705448, 0.704815, -0.056878], [0,0,0,0], [9E9, 9E9, 9E9, 9E9, 9E9, 9E9]];
	VAR robtarget Openhole_2930 := [[451.03, -3.16, 180.92], [-0.046529, 0.705574, 0.704697, -0.058331], [0,0,0,0], [9E9, 9E9, 9E9, 9E9, 9E9, 9E9]];
	VAR robtarget Openhole_2931 := [[456.9, -4.06, 180.09], [-0.023521, 0.706715, 0.703106, -0.075112], [0,0,0,0], [9E9, 9E9, 9E9, 9E9, 9E9, 9E9]];
	VAR robtarget Openhole_2932 := [[457.4, -4.11, 180.03], [-0.021672, 0.706775, 0.702947, -0.076589], [0,0,0,0], [9E9, 9E9, 9E9, 9E9, 9E9, 9E9]];
	VAR robtarget Openhole_2933 := [[458.38, -4.18, 179.89], [-0.01805, 0.706876, 0.702609, -0.079628], [0,0,0,0], [9E9, 9E9, 9E9, 9E9, 9E9, 9E9]];
	VAR robtarget Openhole_2934 := [[459.37, -4.22, 179.75], [-0.01454, 0.706957, 0.702245, -0.082777], [0,0,0,0], [9E9, 9E9, 9E9, 9E9, 9E9, 9E9]];
	VAR robtarget Openhole_2935 := [[459.87, -4.23, 179.68], [-0.012826, 0.70699, 0.702053, -0.08439], [0,0,0,0], [9E9, 9E9, 9E9, 9E9, 9E9, 9E9]];
	VAR robtarget Openhole_2936 := [[460.36, -4.23, 179.61], [-0.011138, 0.707019, 0.701855, -0.086023], [0,0,0,0], [9E9, 9E9, 9E9, 9E9, 9E9, 9E9]];
	VAR robtarget Openhole_2937 := [[464.81, -4, 178.94], [0.003208, 0.7071, 0.699813, -0.1013], [0,0,0,0], [9E9, 9E9, 9E9, 9E9, 9E9, 9E9]];
	VAR robtarget Openhole_2938 := [[473.16, -3.27, 177.57], [0.028952, 0.706514, 0.695045, -0.130048], [0,0,0,0], [9E9, 9E9, 9E9, 9E9, 9E9, 9E9]];
	VAR robtarget Openhole_2939 := [[477.6, -3.15, 176.86], [0.043236, 0.705784, 0.692306, -0.14392], [0,0,0,0], [9E9, 9E9, 9E9, 9E9, 9E9, 9E9]];
	VAR robtarget Openhole_2940 := [[478.1, -3.15, 176.79], [0.044858, 0.705682, 0.691998, -0.145392], [0,0,0,0], [9E9, 9E9, 9E9, 9E9, 9E9, 9E9]];
	VAR robtarget Openhole_2941 := [[484.03, -3.38, 175.96], [0.064771, 0.704134, 0.688308, -0.161962], [0,0,0,0], [9E9, 9E9, 9E9, 9E9, 9E9, 9E9]];
	VAR robtarget Openhole_2942 := [[490.46, -3.99, 175.23], [0.086761, 0.701764, 0.684347, -0.17796], [0,0,0,0], [9E9, 9E9, 9E9, 9E9, 9E9, 9E9]];
	VAR robtarget Openhole_2943 := [[501.83, -5.45, 174.32], [0.124577, 0.696046, 0.677333, -0.203026], [0,0,0,0], [9E9, 9E9, 9E9, 9E9, 9E9, 9E9]];
	VAR robtarget Openhole_2944 := [[503.82, -5.61, 174.15], [0.130603, 0.694941, 0.676013, -0.20738], [0,0,0,0], [9E9, 9E9, 9E9, 9E9, 9E9, 9E9]];
	VAR robtarget Openhole_2945 := [[504.32, -5.62, 174.09], [0.132011, 0.694675, 0.675657, -0.208538], [0,0,0,0], [9E9, 9E9, 9E9, 9E9, 9E9, 9E9]];
	VAR robtarget Openhole_2946 := [[509.32, -5.62, 173.44], [0.183051, 0.683002, 0.683002, -0.183051], [0,0,0,0], [9E9, 9E9, 9E9, 9E9, 9E9, 9E9]];
	VAR robtarget Openhole_2947 := [[536.32, -5.62, 173.36], [0.183051, 0.683002, 0.683002, -0.183051], [0,0,0,0], [9E9, 9E9, 9E9, 9E9, 9E9, 9E9]];
	VAR robtarget Openhole_2948 := [[536.32, -4.67, 172.81], [0.183051, 0.683002, 0.683002, -0.183051], [0,0,0,0], [9E9, 9E9, 9E9, 9E9, 9E9, 9E9]];
	VAR robtarget Openhole_2949 := [[509.32, -4.67, 172.89], [0.183051, 0.683002, 0.683002, -0.183051], [0,0,0,0], [9E9, 9E9, 9E9, 9E9, 9E9, 9E9]];
	VAR robtarget Openhole_2950 := [[504.32, -4.67, 173.58], [0.129262, 0.695192, 0.674813, -0.211251], [0,0,0,0], [9E9, 9E9, 9E9, 9E9, 9E9, 9E9]];
	VAR robtarget Openhole_2951 := [[503.48, -4.58, 173.65], [0.126655, 0.695671, 0.675363, -0.209487], [0,0,0,0], [9E9, 9E9, 9E9, 9E9, 9E9, 9E9]];
	VAR robtarget Openhole_2952 := [[501.51, -4.28, 173.77], [0.120205, 0.696815, 0.676561, -0.205584], [0,0,0,0], [9E9, 9E9, 9E9, 9E9, 9E9, 9E9]];
	VAR robtarget Openhole_2953 := [[494.13, -3.03, 174.28], [0.094931, 0.700705, 0.680941, -0.190577], [0,0,0,0], [9E9, 9E9, 9E9, 9E9, 9E9, 9E9]];
	VAR robtarget Openhole_2954 := [[487.72, -2.18, 174.96], [0.072663, 0.703363, 0.684867, -0.175948], [0,0,0,0], [9E9, 9E9, 9E9, 9E9, 9E9, 9E9]];
	VAR robtarget Openhole_2955 := [[481.8, -1.7, 175.77], [0.052278, 0.705172, 0.688591, -0.160754], [0,0,0,0], [9E9, 9E9, 9E9, 9E9, 9E9, 9E9]];
	VAR robtarget Openhole_2956 := [[476.86, -1.55, 176.55], [0.03568, 0.706206, 0.691716, -0.146727], [0,0,0,0], [9E9, 9E9, 9E9, 9E9, 9E9, 9E9]];
	VAR robtarget Openhole_2957 := [[476.37, -1.55, 176.63], [0.034052, 0.706286, 0.692028, -0.14525], [0,0,0,0], [9E9, 9E9, 9E9, 9E9, 9E9, 9E9]];
	VAR robtarget Openhole_2958 := [[470.95, -1.73, 177.58], [0.016581, 0.706912, 0.695401, -0.128132], [0,0,0,0], [9E9, 9E9, 9E9, 9E9, 9E9, 9E9]];
	VAR robtarget Openhole_2959 := [[462.6, -2.3, 179.05], [-0.009895, 0.707038, 0.700042, -0.099702], [0,0,0,0], [9E9, 9E9, 9E9, 9E9, 9E9, 9E9]];
	VAR robtarget Openhole_2960 := [[461.12, -2.32, 179.29], [-0.014866, 0.70695, 0.700725, -0.094787], [0,0,0,0], [9E9, 9E9, 9E9, 9E9, 9E9, 9E9]];
	VAR robtarget Openhole_2961 := [[460.13, -2.3, 179.44], [-0.018302, 0.70687, 0.701148, -0.091608], [0,0,0,0], [9E9, 9E9, 9E9, 9E9, 9E9, 9E9]];
	VAR robtarget Openhole_2962 := [[459.64, -2.28, 179.52], [-0.020056, 0.706822, 0.701349, -0.09005], [0,0,0,0], [9E9, 9E9, 9E9, 9E9, 9E9, 9E9]];
	VAR robtarget Openhole_2963 := [[455.71, -1.86, 180.13], [-0.03488, 0.706246, 0.702748, -0.078391], [0,0,0,0], [9E9, 9E9, 9E9, 9E9, 9E9, 9E9]];
	VAR robtarget Openhole_2964 := [[455.22, -1.78, 180.21], [-0.0368, 0.706149, 0.702901, -0.077012], [0,0,0,0], [9E9, 9E9, 9E9, 9E9, 9E9, 9E9]];
	VAR robtarget Openhole_2965 := [[452.8, -1.31, 180.59], [-0.04663, 0.705568, 0.703591, -0.070421], [0,0,0,0], [9E9, 9E9, 9E9, 9E9, 9E9, 9E9]];
	VAR robtarget Openhole_2966 := [[452.32, -1.2, 180.67], [-0.048639, 0.705432, 0.703715, -0.069171], [0,0,0,0], [9E9, 9E9, 9E9, 9E9, 9E9, 9E9]];
	VAR robtarget Openhole_2967 := [[451.35, -1, 180.83], [-0.052591, 0.705148, 0.703966, -0.066572], [0,0,0,0], [9E9, 9E9, 9E9, 9E9, 9E9, 9E9]];
	VAR robtarget Openhole_2968 := [[450.86, -0.92, 180.92], [-0.054512, 0.705002, 0.704095, -0.065192], [0,0,0,0], [9E9, 9E9, 9E9, 9E9, 9E9, 9E9]];
	VAR robtarget Openhole_2969 := [[450.37, -0.87, 181], [-0.056351, 0.704858, 0.704231, -0.06371], [0,0,0,0], [9E9, 9E9, 9E9, 9E9, 9E9, 9E9]];
	VAR robtarget Openhole_2970 := [[449.88, -0.83, 181.09], [-0.058145, 0.704712, 0.704368, -0.062171], [0,0,0,0], [9E9, 9E9, 9E9, 9E9, 9E9, 9E9]];
	VAR robtarget Openhole_2971 := [[449.39, -0.83, 181.17], [-0.0598, 0.704574, 0.704515, -0.060482], [0,0,0,0], [9E9, 9E9, 9E9, 9E9, 9E9, 9E9]];
	VAR robtarget Openhole_2972 := [[448.9, -0.86, 181.26], [-0.061392, 0.704437, 0.704663, -0.058737], [0,0,0,0], [9E9, 9E9, 9E9, 9E9, 9E9, 9E9]];
	VAR robtarget Openhole_2973 := [[448.41, -0.92, 181.34], [-0.06283, 0.70431, 0.704817, -0.05686], [0,0,0,0], [9E9, 9E9, 9E9, 9E9, 9E9, 9E9]];
	VAR robtarget Openhole_2974 := [[447.93, -1.01, 181.43], [-0.064179, 0.704188, 0.704971, -0.05492], [0,0,0,0], [9E9, 9E9, 9E9, 9E9, 9E9, 9E9]];
	VAR robtarget Openhole_2975 := [[447.44, -1.11, 181.51], [-0.065469, 0.704069, 0.705122, -0.052937], [0,0,0,0], [9E9, 9E9, 9E9, 9E9, 9E9, 9E9]];
	VAR robtarget Openhole_2976 := [[446.48, -1.34, 181.67], [-0.067964, 0.703833, 0.705413, -0.048914], [0,0,0,0], [9E9, 9E9, 9E9, 9E9, 9E9, 9E9]];
	VAR robtarget Openhole_2977 := [[438.37, -3.6, 182.81], [-0.087546, 0.701666, 0.706974, -0.013685], [0,0,0,0], [9E9, 9E9, 9E9, 9E9, 9E9, 9E9]];
	VAR robtarget Openhole_2978 := [[433.03, -4.74, 183.43], [-0.101226, 0.699824, 0.707058, 0.008281], [0,0,0,0], [9E9, 9E9, 9E9, 9E9, 9E9, 9E9]];
	VAR robtarget Openhole_2979 := [[426.64, -5.75, 184.08], [-0.118226, 0.697153, 0.706334, 0.03306], [0,0,0,0], [9E9, 9E9, 9E9, 9E9, 9E9, 9E9]];
	VAR robtarget Openhole_2980 := [[418.23, -6.67, 184.88], [-0.140885, 0.69293, 0.704242, 0.063588], [0,0,0,0], [9E9, 9E9, 9E9, 9E9, 9E9, 9E9]];
	VAR robtarget Openhole_2981 := [[406.31, -7.48, 185.97], [-0.172244, 0.685808, 0.699547, 0.103122], [0,0,0,0], [9E9, 9E9, 9E9, 9E9, 9E9, 9E9]];
	VAR robtarget Openhole_2982 := [[394.35, -8.14, 186.95], [-0.201027, 0.677929, 0.693251, 0.139296], [0,0,0,0], [9E9, 9E9, 9E9, 9E9, 9E9, 9E9]];
	VAR robtarget Openhole_2983 := [[389.37, -8.14, 187.47], [-0.212867, 0.674305, 0.690443, 0.152605], [0,0,0,0], [9E9, 9E9, 9E9, 9E9, 9E9, 9E9]];
	VAR robtarget Openhole_2984 := [[362.37, -8.14, 187.55], [-0.183051, 0.683002, 0.683002, 0.183051], [0,0,0,0], [9E9, 9E9, 9E9, 9E9, 9E9, 9E9]];
	VAR robtarget Openhole_2985 := [[362.37, -7.26, 188.06], [-0.183051, 0.683002, 0.683002, 0.183051], [0,0,0,0], [9E9, 9E9, 9E9, 9E9, 9E9, 9E9]];
	VAR robtarget Openhole_2986 := [[374.37, -7.26, 188.03], [-0.183051, 0.683002, 0.683002, 0.183051], [0,0,0,0], [9E9, 9E9, 9E9, 9E9, 9E9, 9E9]];
	VAR robtarget Openhole_2987 := [[389.37, -7.26, 187.98], [-0.215327, 0.673524, 0.690996, 0.15008], [0,0,0,0], [9E9, 9E9, 9E9, 9E9, 9E9, 9E9]];
	VAR robtarget Openhole_2988 := [[394.35, -7.26, 187.41], [-0.203559, 0.677173, 0.693763, 0.136721], [0,0,0,0], [9E9, 9E9, 9E9, 9E9, 9E9, 9E9]];
	VAR robtarget Openhole_2989 := [[412.75, -6.11, 185.73], [-0.158528, 0.689107, 0.702662, 0.079161], [0,0,0,0], [9E9, 9E9, 9E9, 9E9, 9E9, 9E9]];
	VAR robtarget Openhole_2990 := [[421.67, -5.25, 184.85], [-0.135112, 0.694078, 0.705486, 0.047849], [0,0,0,0], [9E9, 9E9, 9E9, 9E9, 9E9, 9E9]];
	VAR robtarget Openhole_2991 := [[429.05, -4.16, 184.09], [-0.115814, 0.697558, 0.70683, 0.019796], [0,0,0,0], [9E9, 9E9, 9E9, 9E9, 9E9, 9E9]];
	VAR robtarget Openhole_2992 := [[435.37, -2.86, 183.36], [-0.099805, 0.700028, 0.707082, -0.005926], [0,0,0,0], [9E9, 9E9, 9E9, 9E9, 9E9, 9E9]];
	VAR robtarget Openhole_2993 := [[442.06, -1.02, 182.44], [-0.083814, 0.702122, 0.706246, -0.034871], [0,0,0,0], [9E9, 9E9, 9E9, 9E9, 9E9, 9E9]];
	VAR robtarget Openhole_2994 := [[446.8, 0.36, 181.66], [-0.072458, 0.703385, 0.704917, -0.05561], [0,0,0,0], [9E9, 9E9, 9E9, 9E9, 9E9, 9E9]];
	VAR robtarget Openhole_2995 := [[447.76, 0.61, 181.48], [-0.070062, 0.703627, 0.704584, -0.059673], [0,0,0,0], [9E9, 9E9, 9E9, 9E9, 9E9, 9E9]];
	VAR robtarget Openhole_2996 := [[448.72, 0.81, 181.3], [-0.067477, 0.70388, 0.70424, -0.063612], [0,0,0,0], [9E9, 9E9, 9E9, 9E9, 9E9, 9E9]];
	VAR robtarget Openhole_2997 := [[449.21, 0.87, 181.21], [-0.066004, 0.704019, 0.704071, -0.065448], [0,0,0,0], [9E9, 9E9, 9E9, 9E9, 9E9, 9E9]];
	VAR robtarget Openhole_2998 := [[449.7, 0.9, 181.11], [-0.064452, 0.704163, 0.703905, -0.067219], [0,0,0,0], [9E9, 9E9, 9E9, 9E9, 9E9, 9E9]];
	VAR robtarget Openhole_2999 := [[450.19, 0.88, 181.02], [-0.062708, 0.704321, 0.703751, -0.068804], [0,0,0,0], [9E9, 9E9, 9E9, 9E9, 9E9, 9E9]];
	VAR robtarget Openhole_3000 := [[450.68, 0.85, 180.93], [-0.060938, 0.704476, 0.703598, -0.070355], [0,0,0,0], [9E9, 9E9, 9E9, 9E9, 9E9, 9E9]];
	VAR robtarget Openhole_3001 := [[451.16, 0.77, 180.83], [-0.059051, 0.704637, 0.703456, -0.071765], [0,0,0,0], [9E9, 9E9, 9E9, 9E9, 9E9, 9E9]];
	VAR robtarget Openhole_3002 := [[451.65, 0.69, 180.74], [-0.057117, 0.704796, 0.703317, -0.073109], [0,0,0,0], [9E9, 9E9, 9E9, 9E9, 9E9, 9E9]];
	VAR robtarget Openhole_3003 := [[453.08, 0.32, 180.49], [-0.051048, 0.705262, 0.70293, -0.076745], [0,0,0,0], [9E9, 9E9, 9E9, 9E9, 9E9, 9E9]];
	VAR robtarget Openhole_3004 := [[453.55, 0.19, 180.4], [-0.048987, 0.705408, 0.702803, -0.077896], [0,0,0,0], [9E9, 9E9, 9E9, 9E9, 9E9, 9E9]];
	VAR robtarget Openhole_3005 := [[454.52, -0.01, 180.23], [-0.045034, 0.705671, 0.702512, -0.080476], [0,0,0,0], [9E9, 9E9, 9E9, 9E9, 9E9, 9E9]];
	VAR robtarget Openhole_3006 := [[455.49, -0.16, 180.06], [-0.041204, 0.705905, 0.702192, -0.083229], [0,0,0,0], [9E9, 9E9, 9E9, 9E9, 9E9, 9E9]];
	VAR robtarget Openhole_3007 := [[456.96, -0.33, 179.81], [-0.035634, 0.706208, 0.701663, -0.087574], [0,0,0,0], [9E9, 9E9, 9E9, 9E9, 9E9, 9E9]];
	VAR robtarget Openhole_3008 := [[457.94, -0.41, 179.64], [-0.032016, 0.706382, 0.701282, -0.090575], [0,0,0,0], [9E9, 9E9, 9E9, 9E9, 9E9, 9E9]];
	VAR robtarget Openhole_3009 := [[459.91, -0.49, 179.3], [-0.025, 0.706665, 0.700452, -0.096786], [0,0,0,0], [9E9, 9E9, 9E9, 9E9, 9E9, 9E9]];
	VAR robtarget Openhole_3010 := [[460.9, -0.5, 179.12], [-0.02161, 0.706776, 0.700001, -0.09999], [0,0,0,0], [9E9, 9E9, 9E9, 9E9, 9E9, 9E9]];
	VAR robtarget Openhole_3011 := [[467.28, -0.21, 177.93], [-0.000773, 0.707106, 0.696596, -0.121468], [0,0,0,0], [9E9, 9E9, 9E9, 9E9, 9E9, 9E9]];
	VAR robtarget Openhole_3012 := [[474.15, 0.08, 176.62], [0.021464, 0.706781, 0.692357, -0.143674], [0,0,0,0], [9E9, 9E9, 9E9, 9E9, 9E9, 9E9]];
	VAR robtarget Openhole_3013 := [[475.62, 0.08, 176.35], [0.026358, 0.706615, 0.691414, -0.148146], [0,0,0,0], [9E9, 9E9, 9E9, 9E9, 9E9, 9E9]];
	VAR robtarget Openhole_3014 := [[476.12, 0.08, 176.26], [0.028005, 0.706552, 0.691099, -0.149607], [0,0,0,0], [9E9, 9E9, 9E9, 9E9, 9E9, 9E9]];
	VAR robtarget Openhole_3015 := [[482.02, -0.15, 175.24], [0.048149, 0.705466, 0.687306, -0.166164], [0,0,0,0], [9E9, 9E9, 9E9, 9E9, 9E9, 9E9]];
	VAR robtarget Openhole_3016 := [[487.93, -0.71, 174.37], [0.06877, 0.703755, 0.683554, -0.180981], [0,0,0,0], [9E9, 9E9, 9E9, 9E9, 9E9, 9E9]];
	VAR robtarget Openhole_3017 := [[493.83, -1.55, 173.7], [0.089573, 0.701411, 0.679928, -0.19416], [0,0,0,0], [9E9, 9E9, 9E9, 9E9, 9E9, 9E9]];
	VAR robtarget Openhole_3018 := [[499.22, -2.58, 173.28], [0.108635, 0.698712, 0.676791, -0.204826], [0,0,0,0], [9E9, 9E9, 9E9, 9E9, 9E9, 9E9]];
	VAR robtarget Openhole_3019 := [[503.61, -3.55, 173.09], [0.124001, 0.696149, 0.674344, -0.212745], [0,0,0,0], [9E9, 9E9, 9E9, 9E9, 9E9, 9E9]];
	VAR robtarget Openhole_3020 := [[504.32, -3.66, 173.05], [0.126322, 0.695732, 0.673914, -0.214102], [0,0,0,0], [9E9, 9E9, 9E9, 9E9, 9E9, 9E9]];
	VAR robtarget Openhole_3021 := [[509.32, -3.66, 172.31], [0.183051, 0.683002, 0.683002, -0.183051], [0,0,0,0], [9E9, 9E9, 9E9, 9E9, 9E9, 9E9]];
	VAR robtarget Openhole_3022 := [[536.32, -3.66, 172.22], [0.183051, 0.683002, 0.683002, -0.183051], [0,0,0,0], [9E9, 9E9, 9E9, 9E9, 9E9, 9E9]];
	VAR robtarget Openhole_3023 := [[536.32, -2.79, 171.72], [0.183051, 0.683002, 0.683002, -0.183051], [0,0,0,0], [9E9, 9E9, 9E9, 9E9, 9E9, 9E9]];
	VAR robtarget Openhole_3024 := [[524.32, -2.79, 171.76], [0.183051, 0.683002, 0.683002, -0.183051], [0,0,0,0], [9E9, 9E9, 9E9, 9E9, 9E9, 9E9]];
	VAR robtarget Openhole_3025 := [[509.32, -2.79, 171.81], [0.183051, 0.683002, 0.683002, -0.183051], [0,0,0,0], [9E9, 9E9, 9E9, 9E9, 9E9, 9E9]];
	VAR robtarget Openhole_3026 := [[504.4, -2.79, 172.57], [0.124024, 0.696145, 0.673066, -0.216753], [0,0,0,0], [9E9, 9E9, 9E9, 9E9, 9E9, 9E9]];
	VAR robtarget Openhole_3027 := [[503.83, -2.67, 172.6], [0.122076, 0.696489, 0.67339, -0.215745], [0,0,0,0], [9E9, 9E9, 9E9, 9E9, 9E9, 9E9]];
	VAR robtarget Openhole_3028 := [[498.02, -1.2, 172.83], [0.101022, 0.699853, 0.676485, -0.205836], [0,0,0,0], [9E9, 9E9, 9E9, 9E9, 9E9, 9E9]];
	VAR robtarget Openhole_3029 := [[492.64, -0.16, 173.31], [0.081717, 0.702369, 0.679636, -0.19518], [0,0,0,0], [9E9, 9E9, 9E9, 9E9, 9E9, 9E9]];
	VAR robtarget Openhole_3030 := [[486.76, 0.7, 174.08], [0.060713, 0.704496, 0.683288, -0.181981], [0,0,0,0], [9E9, 9E9, 9E9, 9E9, 9E9, 9E9]];
	VAR robtarget Openhole_3031 := [[480.86, 1.26, 175.02], [0.039935, 0.705978, 0.687067, -0.167148], [0,0,0,0], [9E9, 9E9, 9E9, 9E9, 9E9, 9E9]];
	VAR robtarget Openhole_3032 := [[480.37, 1.3, 175.11], [0.038327, 0.706067, 0.687408, -0.165743], [0,0,0,0], [9E9, 9E9, 9E9, 9E9, 9E9, 9E9]];
	VAR robtarget Openhole_3033 := [[490.33, 1.3, 173.16], [0.070345, 0.703599, 0.680192, -0.193232], [0,0,0,0], [9E9, 9E9, 9E9, 9E9, 9E9, 9E9]];
	VAR robtarget Openhole_3034 := [[490.83, 1.18, 173.11], [0.072049, 0.703427, 0.679875, -0.194345], [0,0,0,0], [9E9, 9E9, 9E9, 9E9, 9E9, 9E9]];
	VAR robtarget Openhole_3035 := [[496.2, 0.2, 172.5], [0.091439, 0.70117, 0.676636, -0.205337], [0,0,0,0], [9E9, 9E9, 9E9, 9E9, 9E9, 9E9]];
	VAR robtarget Openhole_3036 := [[501.06, -0.96, 172.18], [0.109161, 0.69863, 0.673958, -0.213963], [0,0,0,0], [9E9, 9E9, 9E9, 9E9, 9E9, 9E9]];
	VAR robtarget Openhole_3037 := [[502.98, -1.51, 172.14], [0.116289, 0.697479, 0.672993, -0.21698], [0,0,0,0], [9E9, 9E9, 9E9, 9E9, 9E9, 9E9]];
	VAR robtarget Openhole_3038 := [[503.45, -1.68, 172.14], [0.118102, 0.697174, 0.672779, -0.217642], [0,0,0,0], [9E9, 9E9, 9E9, 9E9, 9E9, 9E9]];
	VAR robtarget Openhole_3039 := [[504.32, -1.86, 172.1], [0.121094, 0.696661, 0.672287, -0.219157], [0,0,0,0], [9E9, 9E9, 9E9, 9E9, 9E9, 9E9]];
	VAR robtarget Openhole_3040 := [[509.31, -1.86, 171.27], [0.183051, 0.683002, 0.683002, -0.183051], [0,0,0,0], [9E9, 9E9, 9E9, 9E9, 9E9, 9E9]];
	VAR robtarget Openhole_3041 := [[536.31, -1.86, 171.19], [0.183051, 0.683002, 0.683002, -0.183051], [0,0,0,0], [9E9, 9E9, 9E9, 9E9, 9E9, 9E9]];
	VAR robtarget Openhole_3042 := [[536.31, -1.34, 170.88], [0.183051, 0.683002, 0.683002, -0.183051], [0,0,0,0], [9E9, 9E9, 9E9, 9E9, 9E9, 9E9]];
	VAR robtarget Openhole_3043 := [[509.31, -1.34, 170.97], [0.183051, 0.683002, 0.683002, -0.183051], [0,0,0,0], [9E9, 9E9, 9E9, 9E9, 9E9, 9E9]];
	VAR robtarget Openhole_3044 := [[504.32, -1.34, 171.82], [0.119569, 0.696924, 0.671806, -0.220628], [0,0,0,0], [9E9, 9E9, 9E9, 9E9, 9E9, 9E9]];
	VAR robtarget Openhole_3045 := [[503.61, -1.18, 171.85], [0.117098, 0.697344, 0.672203, -0.219416], [0,0,0,0], [9E9, 9E9, 9E9, 9E9, 9E9, 9E9]];
	VAR robtarget Openhole_3046 := [[499.76, -0.1, 171.99], [0.10287, 0.699584, 0.674183, -0.213254], [0,0,0,0], [9E9, 9E9, 9E9, 9E9, 9E9, 9E9]];
	VAR robtarget Openhole_3047 := [[494.89, 0.95, 172.42], [0.085224, 0.701952, 0.676983, -0.204193], [0,0,0,0], [9E9, 9E9, 9E9, 9E9, 9E9, 9E9]];
	VAR robtarget Openhole_3048 := [[492.93, 1.3, 172.65], [0.078427, 0.702744, 0.67823, -0.200011], [0,0,0,0], [9E9, 9E9, 9E9, 9E9, 9E9, 9E9]];
	VAR robtarget Openhole_3049 := [[445.28, 1.3, 181.98], [-0.080649, 0.702493, 0.705081, -0.053488], [0,0,0,0], [9E9, 9E9, 9E9, 9E9, 9E9, 9E9]];
	VAR robtarget Openhole_3050 := [[444.81, 1.13, 182.06], [-0.081694, 0.702372, 0.705241, -0.051329], [0,0,0,0], [9E9, 9E9, 9E9, 9E9, 9E9, 9E9]];
	VAR robtarget Openhole_3051 := [[436.71, -1.11, 183.36], [-0.101145, 0.699835, 0.70692, -0.016259], [0,0,0,0], [9E9, 9E9, 9E9, 9E9, 9E9, 9E9]];
	VAR robtarget Openhole_3052 := [[429.96, -2.73, 184.22], [-0.117547, 0.697268, 0.707004, 0.012048], [0,0,0,0], [9E9, 9E9, 9E9, 9E9, 9E9, 9E9]];
	VAR robtarget Openhole_3053 := [[423.11, -3.95, 184.99], [-0.134864, 0.694127, 0.706035, 0.038912], [0,0,0,0], [9E9, 9E9, 9E9, 9E9, 9E9, 9E9]];
	VAR robtarget Openhole_3054 := [[415.71, -4.87, 185.77], [-0.153925, 0.69015, 0.70403, 0.065894], [0,0,0,0], [9E9, 9E9, 9E9, 9E9, 9E9, 9E9]];
	VAR robtarget Openhole_3055 := [[405.3, -5.7, 186.84], [-0.180306, 0.683732, 0.699903, 0.100675], [0,0,0,0], [9E9, 9E9, 9E9, 9E9, 9E9, 9E9]];
	VAR robtarget Openhole_3056 := [[394.35, -6.37, 187.88], [-0.20607, 0.676414, 0.694269, 0.134128], [0,0,0,0], [9E9, 9E9, 9E9, 9E9, 9E9, 9E9]];
	VAR robtarget Openhole_3057 := [[389.37, -6.37, 188.49], [-0.217781, 0.672734, 0.69154, 0.147556], [0,0,0,0], [9E9, 9E9, 9E9, 9E9, 9E9, 9E9]];
	VAR robtarget Openhole_3058 := [[362.37, -6.37, 188.57], [-0.183051, 0.683002, 0.683002, 0.183051], [0,0,0,0], [9E9, 9E9, 9E9, 9E9, 9E9, 9E9]];
	VAR robtarget Openhole_3059 := [[362.37, -5.47, 189.1], [-0.183051, 0.683002, 0.683002, 0.183051], [0,0,0,0], [9E9, 9E9, 9E9, 9E9, 9E9, 9E9]];
	VAR robtarget Openhole_3060 := [[389.37, -5.47, 189.01], [-0.220288, 0.671918, 0.692086, 0.144972], [0,0,0,0], [9E9, 9E9, 9E9, 9E9, 9E9, 9E9]];
	VAR robtarget Openhole_3061 := [[394.37, -5.47, 188.36], [-0.208606, 0.675636, 0.694783, 0.131441], [0,0,0,0], [9E9, 9E9, 9E9, 9E9, 9E9, 9E9]];
	VAR robtarget Openhole_3062 := [[410.22, -4.4, 186.69], [-0.170898, 0.686144, 0.702374, 0.081675], [0,0,0,0], [9E9, 9E9, 9E9, 9E9, 9E9, 9E9]];
	VAR robtarget Openhole_3063 := [[418.62, -3.5, 185.78], [-0.149709, 0.691077, 0.705179, 0.052176], [0,0,0,0], [9E9, 9E9, 9E9, 9E9, 9E9, 9E9]];
	VAR robtarget Openhole_3064 := [[425, -2.5, 185.06], [-0.133712, 0.694349, 0.706554, 0.027952], [0,0,0,0], [9E9, 9E9, 9E9, 9E9, 9E9, 9E9]];
	VAR robtarget Openhole_3065 := [[431.79, -1.04, 184.22], [-0.117202, 0.697326, 0.707107, 0.000293], [0,0,0,0], [9E9, 9E9, 9E9, 9E9, 9E9, 9E9]];
	VAR robtarget Openhole_3066 := [[440.43, 1.14, 182.91], [-0.096284, 0.700521, 0.706172, -0.036355], [0,0,0,0], [9E9, 9E9, 9E9, 9E9, 9E9, 9E9]];
	VAR robtarget Openhole_3067 := [[440.9, 1.3, 182.83], [-0.095218, 0.700666, 0.706058, -0.038503], [0,0,0,0], [9E9, 9E9, 9E9, 9E9, 9E9, 9E9]];
	VAR robtarget Openhole_3068 := [[436.08, 1.3, 183.78], [-0.110988, 0.698342, 0.706766, -0.021958], [0,0,0,0], [9E9, 9E9, 9E9, 9E9, 9E9, 9E9]];
	VAR robtarget Openhole_3069 := [[435.6, 1.08, 183.84], [-0.111846, 0.698205, 0.706835, -0.019598], [0,0,0,0], [9E9, 9E9, 9E9, 9E9, 9E9, 9E9]];
	VAR robtarget Openhole_3070 := [[427.41, -0.87, 185.02], [-0.131488, 0.694774, 0.706956, 0.014602], [0,0,0,0], [9E9, 9E9, 9E9, 9E9, 9E9, 9E9]];
	VAR robtarget Openhole_3071 := [[420.58, -2.17, 185.85], [-0.148096, 0.691424, 0.705888, 0.041506], [0,0,0,0], [9E9, 9E9, 9E9, 9E9, 9E9, 9E9]];
	VAR robtarget Openhole_3072 := [[413.19, -3.14, 186.71], [-0.166428, 0.687242, 0.703788, 0.06843], [0,0,0,0], [9E9, 9E9, 9E9, 9E9, 9E9, 9E9]];
	VAR robtarget Openhole_3073 := [[403.3, -3.99, 187.85], [-0.190631, 0.680926, 0.699793, 0.101435], [0,0,0,0], [9E9, 9E9, 9E9, 9E9, 9E9, 9E9]];
	VAR robtarget Openhole_3074 := [[394.36, -4.59, 188.83], [-0.211134, 0.67485, 0.69526, 0.128893], [0,0,0,0], [9E9, 9E9, 9E9, 9E9, 9E9, 9E9]];
	VAR robtarget Openhole_3075 := [[389.37, -4.59, 189.52], [-0.222727, 0.671113, 0.692609, 0.142454], [0,0,0,0], [9E9, 9E9, 9E9, 9E9, 9E9, 9E9]];
	VAR robtarget Openhole_3076 := [[362.37, -4.58, 189.61], [-0.183051, 0.683002, 0.683002, 0.183051], [0,0,0,0], [9E9, 9E9, 9E9, 9E9, 9E9, 9E9]];
	VAR robtarget Openhole_3077 := [[362.37, -3.7, 190.12], [-0.183051, 0.683002, 0.683002, 0.183051], [0,0,0,0], [9E9, 9E9, 9E9, 9E9, 9E9, 9E9]];
	VAR robtarget Openhole_3078 := [[374.37, -3.7, 190.08], [-0.183051, 0.683002, 0.683002, 0.183051], [0,0,0,0], [9E9, 9E9, 9E9, 9E9, 9E9, 9E9]];
	VAR robtarget Openhole_3079 := [[389.37, -3.7, 190.03], [-0.225162, 0.6703, 0.693122, 0.139935], [0,0,0,0], [9E9, 9E9, 9E9, 9E9, 9E9, 9E9]];
	VAR robtarget Openhole_3080 := [[394.37, -3.7, 189.29], [-0.213618, 0.674068, 0.695736, 0.1263], [0,0,0,0], [9E9, 9E9, 9E9, 9E9, 9E9, 9E9]];
	VAR robtarget Openhole_3081 := [[408.73, -2.65, 187.59], [-0.180247, 0.683748, 0.702469, 0.080853], [0,0,0,0], [9E9, 9E9, 9E9, 9E9, 9E9, 9E9]];
	VAR robtarget Openhole_3082 := [[416.62, -1.76, 186.62], [-0.160941, 0.688548, 0.70511, 0.053102], [0,0,0,0], [9E9, 9E9, 9E9, 9E9, 9E9, 9E9]];
	VAR robtarget Openhole_3083 := [[423.48, -0.63, 185.76], [-0.144241, 0.692239, 0.706591, 0.027014], [0,0,0,0], [9E9, 9E9, 9E9, 9E9, 9E9, 9E9]];
	VAR robtarget Openhole_3084 := [[430.74, 0.96, 184.76], [-0.126928, 0.695622, 0.707102, -0.002596], [0,0,0,0], [9E9, 9E9, 9E9, 9E9, 9E9, 9E9]];
	VAR robtarget Openhole_3085 := [[431.22, 1.07, 184.69], [-0.125783, 0.695829, 0.707092, -0.004609], [0,0,0,0], [9E9, 9E9, 9E9, 9E9, 9E9, 9E9]];
	VAR robtarget Openhole_3086 := [[431.7, 1.3, 184.64], [-0.124975, 0.695975, 0.707072, -0.006991], [0,0,0,0], [9E9, 9E9, 9E9, 9E9, 9E9, 9E9]];
	VAR robtarget Openhole_3087 := [[427.8, 1.3, 185.4], [-0.137143, 0.69368, 0.707079, 0.00627], [0,0,0,0], [9E9, 9E9, 9E9, 9E9, 9E9, 9E9]];
	VAR robtarget Openhole_3088 := [[427.32, 1.15, 185.46], [-0.138172, 0.693476, 0.707057, 0.008384], [0,0,0,0], [9E9, 9E9, 9E9, 9E9, 9E9, 9E9]];
	VAR robtarget Openhole_3089 := [[420.52, -0.2, 186.41], [-0.154424, 0.690039, 0.706218, 0.035449], [0,0,0,0], [9E9, 9E9, 9E9, 9E9, 9E9, 9E9]];
	VAR robtarget Openhole_3090 := [[413.15, -1.26, 187.37], [-0.17228, 0.685798, 0.704324, 0.062675], [0,0,0,0], [9E9, 9E9, 9E9, 9E9, 9E9, 9E9]];
	VAR robtarget Openhole_3091 := [[404.27, -2.12, 188.52], [-0.193608, 0.680085, 0.700982, 0.092869], [0,0,0,0], [9E9, 9E9, 9E9, 9E9, 9E9, 9E9]];
	VAR robtarget Openhole_3092 := [[394.37, -2.82, 189.76], [-0.216101, 0.673276, 0.6962, 0.123717], [0,0,0,0], [9E9, 9E9, 9E9, 9E9, 9E9, 9E9]];
	VAR robtarget Openhole_3093 := [[389.37, -2.82, 190.54], [-0.227589, 0.66948, 0.693625, 0.13742], [0,0,0,0], [9E9, 9E9, 9E9, 9E9, 9E9, 9E9]];
	VAR robtarget Openhole_3094 := [[362.38, -2.82, 190.63], [-0.183051, 0.683002, 0.683002, 0.183051], [0,0,0,0], [9E9, 9E9, 9E9, 9E9, 9E9, 9E9]];
	VAR robtarget Openhole_3095 := [[362.38, -1.93, 191.14], [-0.183051, 0.683002, 0.683002, 0.183051], [0,0,0,0], [9E9, 9E9, 9E9, 9E9, 9E9, 9E9]];
	VAR robtarget Openhole_3096 := [[389.38, -1.93, 191.05], [-0.230008, 0.668653, 0.694118, 0.134907], [0,0,0,0], [9E9, 9E9, 9E9, 9E9, 9E9, 9E9]];
	VAR robtarget Openhole_3097 := [[394.37, -1.93, 190.23], [-0.218576, 0.672477, 0.696653, 0.121137], [0,0,0,0], [9E9, 9E9, 9E9, 9E9, 9E9, 9E9]];
	VAR robtarget Openhole_3098 := [[406.73, -1.02, 188.57], [-0.190433, 0.680981, 0.702331, 0.082043], [0,0,0,0], [9E9, 9E9, 9E9, 9E9, 9E9, 9E9]];
	VAR robtarget Openhole_3099 := [[415.1, -0.08, 187.43], [-0.17041, 0.686265, 0.705135, 0.052764], [0,0,0,0], [9E9, 9E9, 9E9, 9E9, 9E9, 9E9]];
	VAR robtarget Openhole_3100 := [[422.43, 1.1, 186.4], [-0.152781, 0.690404, 0.706666, 0.024967], [0,0,0,0], [9E9, 9E9, 9E9, 9E9, 9E9, 9E9]];
	VAR robtarget Openhole_3101 := [[422.92, 1.19, 186.33], [-0.151621, 0.69066, 0.706731, 0.023049], [0,0,0,0], [9E9, 9E9, 9E9, 9E9, 9E9, 9E9]];
	VAR robtarget Openhole_3102 := [[423.41, 1.3, 186.26], [-0.150499, 0.690905, 0.706792, 0.021084], [0,0,0,0], [9E9, 9E9, 9E9, 9E9, 9E9, 9E9]];
	VAR robtarget Openhole_3103 := [[417.57, 1.3, 187.4], [-0.167566, 0.686966, 0.705951, 0.040413], [0,0,0,0], [9E9, 9E9, 9E9, 9E9, 9E9, 9E9]];
	VAR robtarget Openhole_3104 := [[417.07, 1.15, 187.45], [-0.168587, 0.686716, 0.70583, 0.042472], [0,0,0,0], [9E9, 9E9, 9E9, 9E9, 9E9, 9E9]];
	VAR robtarget Openhole_3105 := [[408.73, 0.11, 188.67], [-0.188485, 0.681523, 0.70339, 0.072406], [0,0,0,0], [9E9, 9E9, 9E9, 9E9, 9E9, 9E9]];
	VAR robtarget Openhole_3106 := [[397.87, -0.81, 190.21], [-0.213402, 0.674136, 0.698831, 0.107869], [0,0,0,0], [9E9, 9E9, 9E9, 9E9, 9E9, 9E9]];
	VAR robtarget Openhole_3107 := [[394.38, -1.04, 190.7], [-0.221069, 0.671661, 0.697098, 0.118549], [0,0,0,0], [9E9, 9E9, 9E9, 9E9, 9E9, 9E9]];
	VAR robtarget Openhole_3108 := [[389.38, -1.04, 191.57], [-0.232439, 0.667812, 0.694605, 0.132378], [0,0,0,0], [9E9, 9E9, 9E9, 9E9, 9E9, 9E9]];
	VAR robtarget Openhole_3109 := [[362.42, -1.04, 191.65], [-0.183051, 0.683002, 0.683002, 0.183051], [0,0,0,0], [9E9, 9E9, 9E9, 9E9, 9E9, 9E9]];
	VAR robtarget Openhole_3110 := [[362.42, -1.04, 191.77], [-0.183051, 0.683002, 0.683002, 0.183051], [0,0,0,0], [9E9, 9E9, 9E9, 9E9, 9E9, 9E9]];
	VAR robtarget Openhole_3111 := [[389.38, -1.04, 191.69], [-0.23261, 0.667752, 0.694625, 0.132274], [0,0,0,0], [9E9, 9E9, 9E9, 9E9, 9E9, 9E9]];
	VAR robtarget Openhole_3112 := [[394.38, -1.04, 190.82], [-0.22124, 0.671605, 0.697115, 0.118451], [0,0,0,0], [9E9, 9E9, 9E9, 9E9, 9E9, 9E9]];
	VAR robtarget Openhole_3113 := [[406.26, -0.14, 189.14], [-0.194434, 0.67985, 0.702486, 0.080709], [0,0,0,0], [9E9, 9E9, 9E9, 9E9, 9E9, 9E9]];
	VAR robtarget Openhole_3114 := [[415.11, 0.87, 187.86], [-0.173441, 0.685506, 0.70536, 0.049676], [0,0,0,0], [9E9, 9E9, 9E9, 9E9, 9E9, 9E9]];
	VAR robtarget Openhole_3115 := [[417.07, 1.15, 187.57], [-0.168744, 0.686677, 0.705832, 0.042434], [0,0,0,0], [9E9, 9E9, 9E9, 9E9, 9E9, 9E9]];
	VAR robtarget Openhole_3116 := [[417.57, 1.3, 187.52], [-0.167565, 0.686966, 0.705951, 0.040412], [0,0,0,0], [9E9, 9E9, 9E9, 9E9, 9E9, 9E9]];
	VAR robtarget Openhole_3117 := [[423.41, 1.3, 186.38], [-0.150565, 0.690891, 0.70679, 0.021158], [0,0,0,0], [9E9, 9E9, 9E9, 9E9, 9E9, 9E9]];
	VAR robtarget Openhole_3118 := [[422.92, 1.19, 186.45], [-0.151769, 0.690627, 0.706732, 0.023029], [0,0,0,0], [9E9, 9E9, 9E9, 9E9, 9E9, 9E9]];
	VAR robtarget Openhole_3119 := [[416.08, 0.05, 187.41], [-0.1682, 0.68681, 0.705399, 0.049119], [0,0,0,0], [9E9, 9E9, 9E9, 9E9, 9E9, 9E9]];
	VAR robtarget Openhole_3120 := [[407.72, -0.93, 188.56], [-0.188263, 0.681584, 0.702719, 0.078648], [0,0,0,0], [9E9, 9E9, 9E9, 9E9, 9E9, 9E9]];
	VAR robtarget Openhole_3121 := [[395.86, -1.84, 190.16], [-0.21551, 0.673465, 0.697433, 0.116563], [0,0,0,0], [9E9, 9E9, 9E9, 9E9, 9E9, 9E9]];
	VAR robtarget Openhole_3122 := [[394.37, -1.93, 190.35], [-0.218746, 0.672421, 0.696671, 0.121037], [0,0,0,0], [9E9, 9E9, 9E9, 9E9, 9E9, 9E9]];
	VAR robtarget Openhole_3123 := [[389.38, -1.93, 191.17], [-0.230178, 0.668594, 0.694139, 0.1348], [0,0,0,0], [9E9, 9E9, 9E9, 9E9, 9E9, 9E9]];
	VAR robtarget Openhole_3124 := [[362.38, -1.93, 191.26], [-0.183051, 0.683002, 0.683002, 0.183051], [0,0,0,0], [9E9, 9E9, 9E9, 9E9, 9E9, 9E9]];
	VAR robtarget Openhole_3125 := [[362.38, -2.82, 190.75], [-0.183051, 0.683002, 0.683002, 0.183051], [0,0,0,0], [9E9, 9E9, 9E9, 9E9, 9E9, 9E9]];
	VAR robtarget Openhole_3126 := [[374.38, -2.82, 190.71], [-0.183051, 0.683002, 0.683002, 0.183051], [0,0,0,0], [9E9, 9E9, 9E9, 9E9, 9E9, 9E9]];
	VAR robtarget Openhole_3127 := [[389.38, -2.82, 190.66], [-0.227758, 0.669422, 0.693647, 0.13731], [0,0,0,0], [9E9, 9E9, 9E9, 9E9, 9E9, 9E9]];
	VAR robtarget Openhole_3128 := [[394.37, -2.82, 189.88], [-0.21627, 0.673221, 0.696218, 0.123614], [0,0,0,0], [9E9, 9E9, 9E9, 9E9, 9E9, 9E9]];
	VAR robtarget Openhole_3129 := [[408.22, -1.78, 188.13], [-0.18436, 0.68265, 0.702601, 0.079697], [0,0,0,0], [9E9, 9E9, 9E9, 9E9, 9E9, 9E9]];
	VAR robtarget Openhole_3130 := [[416.11, -0.88, 187.11], [-0.165266, 0.687523, 0.705195, 0.051967], [0,0,0,0], [9E9, 9E9, 9E9, 9E9, 9E9, 9E9]];
	VAR robtarget Openhole_3131 := [[422.95, 0.24, 186.2], [-0.148701, 0.691294, 0.706631, 0.025932], [0,0,0,0], [9E9, 9E9, 9E9, 9E9, 9E9, 9E9]];
	VAR robtarget Openhole_3132 := [[427.32, 1.15, 185.58], [-0.13831, 0.693448, 0.707057, 0.008378], [0,0,0,0], [9E9, 9E9, 9E9, 9E9, 9E9, 9E9]];
	VAR robtarget Openhole_3133 := [[427.8, 1.3, 185.52], [-0.137211, 0.693666, 0.707078, 0.006344], [0,0,0,0], [9E9, 9E9, 9E9, 9E9, 9E9, 9E9]];
	VAR robtarget Openhole_3134 := [[431.7, 1.3, 184.76], [-0.125046, 0.695962, 0.707073, -0.006918], [0,0,0,0], [9E9, 9E9, 9E9, 9E9, 9E9, 9E9]];
	VAR robtarget Openhole_3135 := [[431.22, 1.07, 184.81], [-0.125912, 0.695806, 0.707092, -0.004601], [0,0,0,0], [9E9, 9E9, 9E9, 9E9, 9E9, 9E9]];
	VAR robtarget Openhole_3136 := [[423.96, -0.54, 185.82], [-0.14321, 0.692453, 0.706662, 0.025064], [0,0,0,0], [9E9, 9E9, 9E9, 9E9, 9E9, 9E9]];
	VAR robtarget Openhole_3137 := [[417.11, -1.69, 186.68], [-0.159889, 0.688793, 0.705247, 0.051245], [0,0,0,0], [9E9, 9E9, 9E9, 9E9, 9E9, 9E9]];
	VAR robtarget Openhole_3138 := [[409.23, -2.6, 187.65], [-0.179205, 0.684021, 0.702668, 0.079109], [0,0,0,0], [9E9, 9E9, 9E9, 9E9, 9E9, 9E9]];
	VAR robtarget Openhole_3139 := [[394.87, -3.67, 189.36], [-0.212691, 0.674361, 0.696025, 0.124695], [0,0,0,0], [9E9, 9E9, 9E9, 9E9, 9E9, 9E9]];
	VAR robtarget Openhole_3140 := [[394.37, -3.7, 189.41], [-0.213787, 0.674014, 0.695755, 0.126194], [0,0,0,0], [9E9, 9E9, 9E9, 9E9, 9E9, 9E9]];
	VAR robtarget Openhole_3141 := [[389.37, -3.7, 190.15], [-0.225331, 0.670243, 0.693145, 0.139823], [0,0,0,0], [9E9, 9E9, 9E9, 9E9, 9E9, 9E9]];
	VAR robtarget Openhole_3142 := [[362.37, -3.7, 190.24], [-0.183051, 0.683002, 0.683002, 0.183051], [0,0,0,0], [9E9, 9E9, 9E9, 9E9, 9E9, 9E9]];
	VAR robtarget Openhole_3143 := [[362.37, -4.58, 189.73], [-0.183051, 0.683002, 0.683002, 0.183051], [0,0,0,0], [9E9, 9E9, 9E9, 9E9, 9E9, 9E9]];
	VAR robtarget Openhole_3144 := [[374.37, -4.58, 189.69], [-0.183051, 0.683002, 0.683002, 0.183051], [0,0,0,0], [9E9, 9E9, 9E9, 9E9, 9E9, 9E9]];
	VAR robtarget Openhole_3145 := [[389.37, -4.59, 189.64], [-0.222895, 0.671057, 0.692632, 0.142339], [0,0,0,0], [9E9, 9E9, 9E9, 9E9, 9E9, 9E9]];
	VAR robtarget Openhole_3146 := [[394.36, -4.59, 188.95], [-0.211302, 0.674797, 0.69528, 0.128785], [0,0,0,0], [9E9, 9E9, 9E9, 9E9, 9E9, 9E9]];
	VAR robtarget Openhole_3147 := [[409.73, -3.48, 187.23], [-0.175147, 0.685072, 0.702537, 0.080264], [0,0,0,0], [9E9, 9E9, 9E9, 9E9, 9E9, 9E9]];
	VAR robtarget Openhole_3148 := [[417.63, -2.6, 186.32], [-0.155547, 0.689786, 0.705158, 0.052461], [0,0,0,0], [9E9, 9E9, 9E9, 9E9, 9E9, 9E9]];
	VAR robtarget Openhole_3149 := [[424, -1.56, 185.56], [-0.139858, 0.693138, 0.706543, 0.028221], [0,0,0,0], [9E9, 9E9, 9E9, 9E9, 9E9, 9E9]];
	VAR robtarget Openhole_3150 := [[430.79, -0.09, 184.68], [-0.123524, 0.696234, 0.707106, 0.000639], [0,0,0,0], [9E9, 9E9, 9E9, 9E9, 9E9, 9E9]];
	VAR robtarget Openhole_3151 := [[435.6, 1.08, 183.96], [-0.111963, 0.698186, 0.706836, -0.019574], [0,0,0,0], [9E9, 9E9, 9E9, 9E9, 9E9, 9E9]];
	VAR robtarget Openhole_3152 := [[436.08, 1.3, 183.9], [-0.111065, 0.69833, 0.706768, -0.021889], [0,0,0,0], [9E9, 9E9, 9E9, 9E9, 9E9, 9E9]];
	VAR robtarget Openhole_3153 := [[440.9, 1.3, 182.95], [-0.095299, 0.700656, 0.706061, -0.038436], [0,0,0,0], [9E9, 9E9, 9E9, 9E9, 9E9, 9E9]];
	VAR robtarget Openhole_3154 := [[440.43, 1.14, 183.03], [-0.096387, 0.700507, 0.706174, -0.036314], [0,0,0,0], [9E9, 9E9, 9E9, 9E9, 9E9, 9E9]];
	VAR robtarget Openhole_3155 := [[431.79, -1.04, 184.34], [-0.117323, 0.697306, 0.707107, 0.000295], [0,0,0,0], [9E9, 9E9, 9E9, 9E9, 9E9, 9E9]];
	VAR robtarget Openhole_3156 := [[425, -2.5, 185.18], [-0.133846, 0.694323, 0.706555, 0.027924], [0,0,0,0], [9E9, 9E9, 9E9, 9E9, 9E9, 9E9]];
	VAR robtarget Openhole_3157 := [[418.62, -3.5, 185.9], [-0.149855, 0.691045, 0.705183, 0.052124], [0,0,0,0], [9E9, 9E9, 9E9, 9E9, 9E9, 9E9]];
	VAR robtarget Openhole_3158 := [[410.22, -4.4, 186.81], [-0.171055, 0.686105, 0.702383, 0.081597], [0,0,0,0], [9E9, 9E9, 9E9, 9E9, 9E9, 9E9]];
	VAR robtarget Openhole_3159 := [[394.37, -5.47, 188.48], [-0.208772, 0.675584, 0.694804, 0.13133], [0,0,0,0], [9E9, 9E9, 9E9, 9E9, 9E9, 9E9]];
	VAR robtarget Openhole_3160 := [[389.37, -5.47, 189.13], [-0.220455, 0.671863, 0.69211, 0.144856], [0,0,0,0], [9E9, 9E9, 9E9, 9E9, 9E9, 9E9]];
	VAR robtarget Openhole_3161 := [[362.37, -5.47, 189.22], [-0.183051, 0.683002, 0.683002, 0.183051], [0,0,0,0], [9E9, 9E9, 9E9, 9E9, 9E9, 9E9]];
	VAR robtarget Openhole_3162 := [[362.37, -6.37, 188.69], [-0.183051, 0.683002, 0.683002, 0.183051], [0,0,0,0], [9E9, 9E9, 9E9, 9E9, 9E9, 9E9]];
	VAR robtarget Openhole_3163 := [[374.37, -6.37, 188.66], [-0.183051, 0.683002, 0.683002, 0.183051], [0,0,0,0], [9E9, 9E9, 9E9, 9E9, 9E9, 9E9]];
	VAR robtarget Openhole_3164 := [[389.37, -6.37, 188.61], [-0.217947, 0.67268, 0.691565, 0.147437], [0,0,0,0], [9E9, 9E9, 9E9, 9E9, 9E9, 9E9]];
	VAR robtarget Openhole_3165 := [[394.35, -6.37, 188], [-0.206235, 0.676363, 0.694291, 0.134014], [0,0,0,0], [9E9, 9E9, 9E9, 9E9, 9E9, 9E9]];
	VAR robtarget Openhole_3166 := [[411.75, -5.23, 186.3], [-0.16424, 0.687768, 0.702628, 0.079458], [0,0,0,0], [9E9, 9E9, 9E9, 9E9, 9E9, 9E9]];
	VAR robtarget Openhole_3167 := [[420.16, -4.36, 185.42], [-0.142593, 0.69258, 0.705345, 0.049888], [0,0,0,0], [9E9, 9E9, 9E9, 9E9, 9E9, 9E9]];
	VAR robtarget Openhole_3168 := [[427.03, -3.3, 184.68], [-0.125015, 0.695968, 0.706709, 0.023724], [0,0,0,0], [9E9, 9E9, 9E9, 9E9, 9E9, 9E9]];
	VAR robtarget Openhole_3169 := [[432.87, -2.08, 183.99], [-0.110536, 0.698414, 0.707107, 0.000052], [0,0,0,0], [9E9, 9E9, 9E9, 9E9, 9E9, 9E9]];
	VAR robtarget Openhole_3170 := [[441.01, 0.05, 182.83], [-0.090904, 0.701239, 0.706252, -0.034753], [0,0,0,0], [9E9, 9E9, 9E9, 9E9, 9E9, 9E9]];
	VAR robtarget Openhole_3171 := [[444.81, 1.13, 182.18], [-0.081783, 0.702361, 0.705246, -0.051272], [0,0,0,0], [9E9, 9E9, 9E9, 9E9, 9E9, 9E9]];
	VAR robtarget Openhole_3172 := [[445.28, 1.3, 182.1], [-0.080728, 0.702483, 0.705086, -0.053419], [0,0,0,0], [9E9, 9E9, 9E9, 9E9, 9E9, 9E9]];
	VAR robtarget Openhole_3173 := [[492.93, 1.3, 172.77], [0.078359, 0.702752, 0.678246, -0.199954], [0,0,0,0], [9E9, 9E9, 9E9, 9E9, 9E9, 9E9]];
	VAR robtarget Openhole_3174 := [[497.82, 0.35, 172.26], [0.095879, 0.700576, 0.675322, -0.209621], [0,0,0,0], [9E9, 9E9, 9E9, 9E9, 9E9, 9E9]];
	VAR robtarget Openhole_3175 := [[502.17, -0.75, 172], [0.111842, 0.698206, 0.672968, -0.217059], [0,0,0,0], [9E9, 9E9, 9E9, 9E9, 9E9, 9E9]];
	VAR robtarget Openhole_3176 := [[503.61, -1.18, 171.97], [0.117194, 0.697327, 0.672259, -0.219244], [0,0,0,0], [9E9, 9E9, 9E9, 9E9, 9E9, 9E9]];
	VAR robtarget Openhole_3177 := [[504.32, -1.34, 171.94], [0.119668, 0.696907, 0.671862, -0.220457], [0,0,0,0], [9E9, 9E9, 9E9, 9E9, 9E9, 9E9]];
	VAR robtarget Openhole_3178 := [[509.31, -1.34, 171.09], [0.183051, 0.683002, 0.683002, -0.183051], [0,0,0,0], [9E9, 9E9, 9E9, 9E9, 9E9, 9E9]];
	VAR robtarget Openhole_3179 := [[536.31, -1.34, 171], [0.183051, 0.683002, 0.683002, -0.183051], [0,0,0,0], [9E9, 9E9, 9E9, 9E9, 9E9, 9E9]];
	VAR robtarget Openhole_3180 := [[536.32, -1.86, 171.31], [0.183051, 0.683002, 0.683002, -0.183051], [0,0,0,0], [9E9, 9E9, 9E9, 9E9, 9E9, 9E9]];
	VAR robtarget Openhole_3181 := [[509.32, -1.86, 171.39], [0.183051, 0.683002, 0.683002, -0.183051], [0,0,0,0], [9E9, 9E9, 9E9, 9E9, 9E9, 9E9]];
	VAR robtarget Openhole_3182 := [[504.32, -1.86, 172.22], [0.121194, 0.696643, 0.672343, -0.218986], [0,0,0,0], [9E9, 9E9, 9E9, 9E9, 9E9, 9E9]];
	VAR robtarget Openhole_3183 := [[503.45, -1.68, 172.26], [0.1182, 0.697158, 0.672834, -0.217472], [0,0,0,0], [9E9, 9E9, 9E9, 9E9, 9E9, 9E9]];
	VAR robtarget Openhole_3184 := [[502.98, -1.51, 172.26], [0.116386, 0.697463, 0.673048, -0.216809], [0,0,0,0], [9E9, 9E9, 9E9, 9E9, 9E9, 9E9]];
	VAR robtarget Openhole_3185 := [[498.64, -0.34, 172.43], [0.100376, 0.699946, 0.675312, -0.20965], [0,0,0,0], [9E9, 9E9, 9E9, 9E9, 9E9, 9E9]];
	VAR robtarget Openhole_3186 := [[493.76, 0.68, 172.87], [0.082692, 0.702255, 0.678132, -0.200343], [0,0,0,0], [9E9, 9E9, 9E9, 9E9, 9E9, 9E9]];
	VAR robtarget Openhole_3187 := [[490.83, 1.18, 173.23], [0.072113, 0.70342, 0.679923, -0.194178], [0,0,0,0], [9E9, 9E9, 9E9, 9E9, 9E9, 9E9]];
	VAR robtarget Openhole_3188 := [[490.33, 1.3, 173.28], [0.070233, 0.70361, 0.680219, -0.193138], [0,0,0,0], [9E9, 9E9, 9E9, 9E9, 9E9, 9E9]];
	VAR robtarget Openhole_3189 := [[480.37, 1.3, 175.23], [0.038255, 0.706071, 0.687423, -0.16568], [0,0,0,0], [9E9, 9E9, 9E9, 9E9, 9E9, 9E9]];
	VAR robtarget Openhole_3190 := [[486.26, 0.75, 174.27], [0.059021, 0.704639, 0.683642, -0.180648], [0,0,0,0], [9E9, 9E9, 9E9, 9E9, 9E9, 9E9]];
	VAR robtarget Openhole_3191 := [[492.15, -0.08, 173.49], [0.080039, 0.702562, 0.679982, -0.193971], [0,0,0,0], [9E9, 9E9, 9E9, 9E9, 9E9, 9E9]];
	VAR robtarget Openhole_3192 := [[497.53, -1.09, 172.98], [0.09935, 0.700093, 0.676811, -0.204761], [0,0,0,0], [9E9, 9E9, 9E9, 9E9, 9E9, 9E9]];
	VAR robtarget Openhole_3193 := [[502.87, -2.42, 172.74], [0.118715, 0.69707, 0.673951, -0.213986], [0,0,0,0], [9E9, 9E9, 9E9, 9E9, 9E9, 9E9]];
	VAR robtarget Openhole_3194 := [[503.83, -2.67, 172.72], [0.122178, 0.696471, 0.673444, -0.215575], [0,0,0,0], [9E9, 9E9, 9E9, 9E9, 9E9, 9E9]];
	VAR robtarget Openhole_3195 := [[504.4, -2.79, 172.69], [0.124127, 0.696127, 0.673121, -0.216584], [0,0,0,0], [9E9, 9E9, 9E9, 9E9, 9E9, 9E9]];
	VAR robtarget Openhole_3196 := [[509.32, -2.79, 171.93], [0.183051, 0.683002, 0.683002, -0.183051], [0,0,0,0], [9E9, 9E9, 9E9, 9E9, 9E9, 9E9]];
	VAR robtarget Openhole_3197 := [[536.32, -2.79, 171.84], [0.183051, 0.683002, 0.683002, -0.183051], [0,0,0,0], [9E9, 9E9, 9E9, 9E9, 9E9, 9E9]];
	VAR robtarget Openhole_3198 := [[536.32, -3.66, 172.34], [0.183051, 0.683002, 0.683002, -0.183051], [0,0,0,0], [9E9, 9E9, 9E9, 9E9, 9E9, 9E9]];
	VAR robtarget Openhole_3199 := [[509.32, -3.66, 172.43], [0.183051, 0.683002, 0.683002, -0.183051], [0,0,0,0], [9E9, 9E9, 9E9, 9E9, 9E9, 9E9]];
	VAR robtarget Openhole_3200 := [[504.32, -3.66, 173.17], [0.126428, 0.695713, 0.673968, -0.213933], [0,0,0,0], [9E9, 9E9, 9E9, 9E9, 9E9, 9E9]];
	VAR robtarget Openhole_3201 := [[503.61, -3.55, 173.21], [0.124106, 0.696131, 0.674397, -0.212576], [0,0,0,0], [9E9, 9E9, 9E9, 9E9, 9E9, 9E9]];
	VAR robtarget Openhole_3202 := [[496.78, -2.08, 173.56], [0.100057, 0.699992, 0.678236, -0.199991], [0,0,0,0], [9E9, 9E9, 9E9, 9E9, 9E9, 9E9]];
	VAR robtarget Openhole_3203 := [[490.89, -1.1, 174.13], [0.079239, 0.702653, 0.681767, -0.187601], [0,0,0,0], [9E9, 9E9, 9E9, 9E9, 9E9, 9E9]];
	VAR robtarget Openhole_3204 := [[484.49, -0.34, 174.98], [0.056741, 0.704827, 0.685769, -0.172398], [0,0,0,0], [9E9, 9E9, 9E9, 9E9, 9E9, 9E9]];
	VAR robtarget Openhole_3205 := [[478.08, 0.04, 176.02], [0.034669, 0.706256, 0.689868, -0.155185], [0,0,0,0], [9E9, 9E9, 9E9, 9E9, 9E9, 9E9]];
	VAR robtarget Openhole_3206 := [[475.62, 0.08, 176.47], [0.026382, 0.706614, 0.691445, -0.148001], [0,0,0,0], [9E9, 9E9, 9E9, 9E9, 9E9, 9E9]];
	VAR robtarget Openhole_3207 := [[475.13, 0.08, 176.56], [0.024745, 0.706674, 0.69176, -0.146521], [0,0,0,0], [9E9, 9E9, 9E9, 9E9, 9E9, 9E9]];
	VAR robtarget Openhole_3208 := [[468.75, -0.12, 177.77], [0.003927, 0.707096, 0.695743, -0.12626], [0,0,0,0], [9E9, 9E9, 9E9, 9E9, 9E9, 9E9]];
	VAR robtarget Openhole_3209 := [[461.39, -0.49, 179.15], [-0.019973, 0.706825, 0.699782, -0.101511], [0,0,0,0], [9E9, 9E9, 9E9, 9E9, 9E9, 9E9]];
	VAR robtarget Openhole_3210 := [[460.9, -0.5, 179.24], [-0.021635, 0.706776, 0.700017, -0.099884], [0,0,0,0], [9E9, 9E9, 9E9, 9E9, 9E9, 9E9]];
	VAR robtarget Openhole_3211 := [[459.91, -0.49, 179.42], [-0.02503, 0.706664, 0.700466, -0.096682], [0,0,0,0], [9E9, 9E9, 9E9, 9E9, 9E9, 9E9]];
	VAR robtarget Openhole_3212 := [[457.94, -0.41, 179.76], [-0.032052, 0.70638, 0.701294, -0.090477], [0,0,0,0], [9E9, 9E9, 9E9, 9E9, 9E9, 9E9]];
	VAR robtarget Openhole_3213 := [[456.96, -0.33, 179.93], [-0.035674, 0.706206, 0.701675, -0.087479], [0,0,0,0], [9E9, 9E9, 9E9, 9E9, 9E9, 9E9]];
	VAR robtarget Openhole_3214 := [[455.49, -0.16, 180.18], [-0.04125, 0.705903, 0.702202, -0.083139], [0,0,0,0], [9E9, 9E9, 9E9, 9E9, 9E9, 9E9]];
	VAR robtarget Openhole_3215 := [[454.52, -0.01, 180.35], [-0.045085, 0.705668, 0.702522, -0.080388], [0,0,0,0], [9E9, 9E9, 9E9, 9E9, 9E9, 9E9]];
	VAR robtarget Openhole_3216 := [[453.55, 0.19, 180.52], [-0.049042, 0.705404, 0.702813, -0.077811], [0,0,0,0], [9E9, 9E9, 9E9, 9E9, 9E9, 9E9]];
	VAR robtarget Openhole_3217 := [[453.08, 0.32, 180.61], [-0.051105, 0.705258, 0.702939, -0.076661], [0,0,0,0], [9E9, 9E9, 9E9, 9E9, 9E9, 9E9]];
	VAR robtarget Openhole_3218 := [[451.65, 0.69, 180.86], [-0.05718, 0.704791, 0.703326, -0.073029], [0,0,0,0], [9E9, 9E9, 9E9, 9E9, 9E9, 9E9]];
	VAR robtarget Openhole_3219 := [[451.16, 0.77, 180.95], [-0.059117, 0.704631, 0.703464, -0.071686], [0,0,0,0], [9E9, 9E9, 9E9, 9E9, 9E9, 9E9]];
	VAR robtarget Openhole_3220 := [[450.68, 0.85, 181.05], [-0.061006, 0.70447, 0.703606, -0.070277], [0,0,0,0], [9E9, 9E9, 9E9, 9E9, 9E9, 9E9]];
	VAR robtarget Openhole_3221 := [[450.19, 0.88, 181.14], [-0.062778, 0.704315, 0.703759, -0.068728], [0,0,0,0], [9E9, 9E9, 9E9, 9E9, 9E9, 9E9]];
	VAR robtarget Openhole_3222 := [[449.7, 0.9, 181.23], [-0.064523, 0.704157, 0.703912, -0.067145], [0,0,0,0], [9E9, 9E9, 9E9, 9E9, 9E9, 9E9]];
	VAR robtarget Openhole_3223 := [[449.21, 0.87, 181.33], [-0.066077, 0.704013, 0.704078, -0.065376], [0,0,0,0], [9E9, 9E9, 9E9, 9E9, 9E9, 9E9]];
	VAR robtarget Openhole_3224 := [[448.72, 0.81, 181.42], [-0.067551, 0.703873, 0.704246, -0.063542], [0,0,0,0], [9E9, 9E9, 9E9, 9E9, 9E9, 9E9]];
	VAR robtarget Openhole_3225 := [[447.76, 0.61, 181.6], [-0.070139, 0.70362, 0.70459, -0.059607], [0,0,0,0], [9E9, 9E9, 9E9, 9E9, 9E9, 9E9]];
	VAR robtarget Openhole_3226 := [[446.8, 0.36, 181.78], [-0.072538, 0.703376, 0.704922, -0.055548], [0,0,0,0], [9E9, 9E9, 9E9, 9E9, 9E9, 9E9]];
	VAR robtarget Openhole_3227 := [[438.73, -1.98, 183.04], [-0.091801, 0.701122, 0.706816, -0.020283], [0,0,0,0], [9E9, 9E9, 9E9, 9E9, 9E9, 9E9]];
	VAR robtarget Openhole_3228 := [[433.43, -3.29, 183.71], [-0.104758, 0.699304, 0.707104, 0.002107], [0,0,0,0], [9E9, 9E9, 9E9, 9E9, 9E9, 9E9]];
	VAR robtarget Openhole_3229 := [[427.08, -4.48, 184.42], [-0.121047, 0.696669, 0.706575, 0.027406], [0,0,0,0], [9E9, 9E9, 9E9, 9E9, 9E9, 9E9]];
	VAR robtarget Openhole_3230 := [[419.69, -5.48, 185.17], [-0.140456, 0.693017, 0.704966, 0.054976], [0,0,0,0], [9E9, 9E9, 9E9, 9E9, 9E9, 9E9]];
	VAR robtarget Openhole_3231 := [[409.77, -6.33, 186.14], [-0.166372, 0.687256, 0.701486, 0.08898], [0,0,0,0], [9E9, 9E9, 9E9, 9E9, 9E9, 9E9]];
	VAR robtarget Openhole_3232 := [[394.35, -7.26, 187.53], [-0.203724, 0.677124, 0.693786, 0.136605], [0,0,0,0], [9E9, 9E9, 9E9, 9E9, 9E9, 9E9]];
	VAR robtarget Openhole_3233 := [[389.37, -7.26, 188.1], [-0.215492, 0.673471, 0.691023, 0.149958], [0,0,0,0], [9E9, 9E9, 9E9, 9E9, 9E9, 9E9]];
	VAR robtarget Openhole_3234 := [[362.37, -7.26, 188.18], [-0.183051, 0.683002, 0.683002, 0.183051], [0,0,0,0], [9E9, 9E9, 9E9, 9E9, 9E9, 9E9]];
	VAR robtarget Openhole_3235 := [[362.37, -8.14, 187.67], [-0.183051, 0.683002, 0.683002, 0.183051], [0,0,0,0], [9E9, 9E9, 9E9, 9E9, 9E9, 9E9]];
	VAR robtarget Openhole_3236 := [[374.37, -8.14, 187.64], [-0.183051, 0.683002, 0.683002, 0.183051], [0,0,0,0], [9E9, 9E9, 9E9, 9E9, 9E9, 9E9]];
	VAR robtarget Openhole_3237 := [[389.37, -8.14, 187.59], [-0.213031, 0.674253, 0.690471, 0.152481], [0,0,0,0], [9E9, 9E9, 9E9, 9E9, 9E9, 9E9]];
	VAR robtarget Openhole_3238 := [[394.35, -8.14, 187.07], [-0.20119, 0.677881, 0.693275, 0.139177], [0,0,0,0], [9E9, 9E9, 9E9, 9E9, 9E9, 9E9]];
	VAR robtarget Openhole_3239 := [[411.28, -7.19, 185.64], [-0.159538, 0.688874, 0.70173, 0.087035], [0,0,0,0], [9E9, 9E9, 9E9, 9E9, 9E9, 9E9]];
	VAR robtarget Openhole_3240 := [[421.2, -6.39, 184.73], [-0.133008, 0.694485, 0.705117, 0.053008], [0,0,0,0], [9E9, 9E9, 9E9, 9E9, 9E9, 9E9]];
	VAR robtarget Openhole_3241 := [[429.6, -5.33, 183.91], [-0.110396, 0.698436, 0.706771, 0.021779], [0,0,0,0], [9E9, 9E9, 9E9, 9E9, 9E9, 9E9]];
	VAR robtarget Openhole_3242 := [[435.95, -4.17, 183.22], [-0.093731, 0.700867, 0.707098, -0.003566], [0,0,0,0], [9E9, 9E9, 9E9, 9E9, 9E9, 9E9]];
	VAR robtarget Openhole_3243 := [[441.25, -2.83, 182.56], [-0.080656, 0.702492, 0.706627, -0.026043], [0,0,0,0], [9E9, 9E9, 9E9, 9E9, 9E9, 9E9]];
	VAR robtarget Openhole_3244 := [[446.48, -1.34, 181.79], [-0.068039, 0.703826, 0.705417, -0.04886], [0,0,0,0], [9E9, 9E9, 9E9, 9E9, 9E9, 9E9]];
	VAR robtarget Openhole_3245 := [[447.44, -1.11, 181.63], [-0.065541, 0.704063, 0.705127, -0.052878], [0,0,0,0], [9E9, 9E9, 9E9, 9E9, 9E9, 9E9]];
	VAR robtarget Openhole_3246 := [[447.93, -1.01, 181.55], [-0.06425, 0.704182, 0.704976, -0.054859], [0,0,0,0], [9E9, 9E9, 9E9, 9E9, 9E9, 9E9]];
	VAR robtarget Openhole_3247 := [[448.41, -0.92, 181.46], [-0.0629, 0.704304, 0.704822, -0.056797], [0,0,0,0], [9E9, 9E9, 9E9, 9E9, 9E9, 9E9]];
	VAR robtarget Openhole_3248 := [[448.9, -0.86, 181.38], [-0.06146, 0.704431, 0.704668, -0.058672], [0,0,0,0], [9E9, 9E9, 9E9, 9E9, 9E9, 9E9]];
	VAR robtarget Openhole_3249 := [[449.39, -0.83, 181.29], [-0.059867, 0.704568, 0.704521, -0.060415], [0,0,0,0], [9E9, 9E9, 9E9, 9E9, 9E9, 9E9]];
	VAR robtarget Openhole_3250 := [[449.88, -0.83, 181.21], [-0.05821, 0.704707, 0.704374, -0.062102], [0,0,0,0], [9E9, 9E9, 9E9, 9E9, 9E9, 9E9]];
	VAR robtarget Openhole_3251 := [[450.37, -0.87, 181.12], [-0.056414, 0.704853, 0.704237, -0.06364], [0,0,0,0], [9E9, 9E9, 9E9, 9E9, 9E9, 9E9]];
	VAR robtarget Openhole_3252 := [[450.86, -0.92, 181.04], [-0.054572, 0.704998, 0.704102, -0.06512], [0,0,0,0], [9E9, 9E9, 9E9, 9E9, 9E9, 9E9]];
	VAR robtarget Openhole_3253 := [[451.35, -1, 180.95], [-0.05265, 0.705144, 0.703973, -0.066499], [0,0,0,0], [9E9, 9E9, 9E9, 9E9, 9E9, 9E9]];
	VAR robtarget Openhole_3254 := [[452.32, -1.2, 180.79], [-0.048693, 0.705428, 0.703723, -0.069095], [0,0,0,0], [9E9, 9E9, 9E9, 9E9, 9E9, 9E9]];
	VAR robtarget Openhole_3255 := [[452.8, -1.31, 180.71], [-0.046682, 0.705564, 0.703599, -0.070344], [0,0,0,0], [9E9, 9E9, 9E9, 9E9, 9E9, 9E9]];
	VAR robtarget Openhole_3256 := [[455.22, -1.78, 180.33], [-0.036842, 0.706146, 0.70291, -0.076928], [0,0,0,0], [9E9, 9E9, 9E9, 9E9, 9E9, 9E9]];
	VAR robtarget Openhole_3257 := [[459.15, -2.25, 179.72], [-0.021864, 0.706769, 0.701556, -0.088424], [0,0,0,0], [9E9, 9E9, 9E9, 9E9, 9E9, 9E9]];
	VAR robtarget Openhole_3258 := [[459.64, -2.28, 179.64], [-0.020079, 0.706822, 0.701362, -0.089953], [0,0,0,0], [9E9, 9E9, 9E9, 9E9, 9E9, 9E9]];
	VAR robtarget Openhole_3259 := [[460.13, -2.3, 179.56], [-0.018323, 0.706869, 0.70116, -0.091509], [0,0,0,0], [9E9, 9E9, 9E9, 9E9, 9E9, 9E9]];
	VAR robtarget Openhole_3260 := [[461.12, -2.32, 179.41], [-0.014884, 0.70695, 0.700739, -0.094686], [0,0,0,0], [9E9, 9E9, 9E9, 9E9, 9E9, 9E9]];
	VAR robtarget Openhole_3261 := [[466.05, -2.11, 178.58], [0.001206, 0.707106, 0.698288, -0.111326], [0,0,0,0], [9E9, 9E9, 9E9, 9E9, 9E9, 9E9]];
	VAR robtarget Openhole_3262 := [[473.41, -1.61, 177.26], [0.02444, 0.706684, 0.69391, -0.135975], [0,0,0,0], [9E9, 9E9, 9E9, 9E9, 9E9, 9E9]];
	VAR robtarget Openhole_3263 := [[476.86, -1.55, 176.67], [0.035714, 0.706204, 0.691747, -0.146583], [0,0,0,0], [9E9, 9E9, 9E9, 9E9, 9E9, 9E9]];
	VAR robtarget Openhole_3264 := [[477.35, -1.55, 176.59], [0.037351, 0.70612, 0.691435, -0.148046], [0,0,0,0], [9E9, 9E9, 9E9, 9E9, 9E9, 9E9]];
	VAR robtarget Openhole_3265 := [[483.28, -1.79, 175.67], [0.05739, 0.704774, 0.687691, -0.164565], [0,0,0,0], [9E9, 9E9, 9E9, 9E9, 9E9, 9E9]];
	VAR robtarget Openhole_3266 := [[489.2, -2.35, 174.9], [0.077874, 0.702806, 0.683991, -0.179323], [0,0,0,0], [9E9, 9E9, 9E9, 9E9, 9E9, 9E9]];
	VAR robtarget Openhole_3267 := [[496.1, -3.34, 174.24], [0.10183, 0.699736, 0.679805, -0.19459], [0,0,0,0], [9E9, 9E9, 9E9, 9E9, 9E9, 9E9]];
	VAR robtarget Openhole_3268 := [[501.51, -4.28, 173.89], [0.120309, 0.696797, 0.676612, -0.205417], [0,0,0,0], [9E9, 9E9, 9E9, 9E9, 9E9, 9E9]];
	VAR robtarget Openhole_3269 := [[503.48, -4.58, 173.77], [0.126762, 0.695652, 0.675415, -0.209319], [0,0,0,0], [9E9, 9E9, 9E9, 9E9, 9E9, 9E9]];
	VAR robtarget Openhole_3270 := [[504.32, -4.67, 173.7], [0.129371, 0.695171, 0.674866, -0.211083], [0,0,0,0], [9E9, 9E9, 9E9, 9E9, 9E9, 9E9]];
	VAR robtarget Openhole_3271 := [[509.32, -4.67, 173.01], [0.183051, 0.683002, 0.683002, -0.183051], [0,0,0,0], [9E9, 9E9, 9E9, 9E9, 9E9, 9E9]];
	VAR robtarget Openhole_3272 := [[536.32, -4.67, 172.93], [0.183051, 0.683002, 0.683002, -0.183051], [0,0,0,0], [9E9, 9E9, 9E9, 9E9, 9E9, 9E9]];
	VAR robtarget Openhole_3273 := [[536.32, -5.62, 173.48], [0.183051, 0.683002, 0.683002, -0.183051], [0,0,0,0], [9E9, 9E9, 9E9, 9E9, 9E9, 9E9]];
	VAR robtarget Openhole_3274 := [[524.32, -5.62, 173.51], [0.183051, 0.683002, 0.683002, -0.183051], [0,0,0,0], [9E9, 9E9, 9E9, 9E9, 9E9, 9E9]];
	VAR robtarget Openhole_3275 := [[509.32, -5.62, 173.56], [0.183051, 0.683002, 0.683002, -0.183051], [0,0,0,0], [9E9, 9E9, 9E9, 9E9, 9E9, 9E9]];
	VAR robtarget Openhole_3276 := [[504.32, -5.62, 174.21], [0.132123, 0.694654, 0.675708, -0.208372], [0,0,0,0], [9E9, 9E9, 9E9, 9E9, 9E9, 9E9]];
	VAR robtarget Openhole_3277 := [[503.82, -5.61, 174.27], [0.130714, 0.69492, 0.676064, -0.207214], [0,0,0,0], [9E9, 9E9, 9E9, 9E9, 9E9, 9E9]];
	VAR robtarget Openhole_3278 := [[498.86, -5.11, 174.67], [0.115216, 0.697657, 0.679271, -0.196446], [0,0,0,0], [9E9, 9E9, 9E9, 9E9, 9E9, 9E9]];
	VAR robtarget Openhole_3279 := [[489.97, -3.94, 175.4], [0.085146, 0.701962, 0.68469, -0.176635], [0,0,0,0], [9E9, 9E9, 9E9, 9E9, 9E9, 9E9]];
	VAR robtarget Openhole_3280 := [[483.54, -3.35, 176.14], [0.063154, 0.704281, 0.688651, -0.160498], [0,0,0,0], [9E9, 9E9, 9E9, 9E9, 9E9, 9E9]];
	VAR robtarget Openhole_3281 := [[478.1, -3.15, 176.91], [0.044903, 0.70568, 0.692028, -0.145249], [0,0,0,0], [9E9, 9E9, 9E9, 9E9, 9E9, 9E9]];
	VAR robtarget Openhole_3282 := [[477.6, -3.15, 176.98], [0.043279, 0.705781, 0.692335, -0.143778], [0,0,0,0], [9E9, 9E9, 9E9, 9E9, 9E9, 9E9]];
	VAR robtarget Openhole_3283 := [[477.11, -3.15, 177.06], [0.041656, 0.705879, 0.69264, -0.142299], [0,0,0,0], [9E9, 9E9, 9E9, 9E9, 9E9, 9E9]];
	VAR robtarget Openhole_3284 := [[471.68, -3.36, 177.93], [0.024353, 0.706687, 0.695962, -0.12505], [0,0,0,0], [9E9, 9E9, 9E9, 9E9, 9E9, 9E9]];
	VAR robtarget Openhole_3285 := [[462.34, -4.17, 179.44], [-0.004613, 0.707092, 0.701014, -0.092624], [0,0,0,0], [9E9, 9E9, 9E9, 9E9, 9E9, 9E9]];
	VAR robtarget Openhole_3286 := [[459.87, -4.23, 179.8], [-0.012841, 0.70699, 0.702064, -0.084299], [0,0,0,0], [9E9, 9E9, 9E9, 9E9, 9E9, 9E9]];
	VAR robtarget Openhole_3287 := [[459.37, -4.22, 179.87], [-0.014556, 0.706957, 0.702256, -0.082687], [0,0,0,0], [9E9, 9E9, 9E9, 9E9, 9E9, 9E9]];
	VAR robtarget Openhole_3288 := [[458.38, -4.18, 180.01], [-0.01807, 0.706876, 0.702619, -0.079541], [0,0,0,0], [9E9, 9E9, 9E9, 9E9, 9E9, 9E9]];
	VAR robtarget Openhole_3289 := [[457.4, -4.11, 180.15], [-0.021696, 0.706774, 0.702956, -0.076505], [0,0,0,0], [9E9, 9E9, 9E9, 9E9, 9E9, 9E9]];
	VAR robtarget Openhole_3290 := [[452.98, -3.48, 180.76], [-0.038865, 0.706038, 0.704222, -0.063809], [0,0,0,0], [9E9, 9E9, 9E9, 9E9, 9E9, 9E9]];
	VAR robtarget Openhole_3291 := [[451.03, -3.16, 181.04], [-0.04658, 0.705571, 0.704702, -0.058266], [0,0,0,0], [9E9, 9E9, 9E9, 9E9, 9E9, 9E9]];
	VAR robtarget Openhole_3292 := [[450.54, -3.1, 181.12], [-0.04846, 0.705444, 0.704821, -0.056815], [0,0,0,0], [9E9, 9E9, 9E9, 9E9, 9E9, 9E9]];
	VAR robtarget Openhole_3293 := [[449.55, -3.01, 181.27], [-0.052109, 0.705184, 0.705059, -0.053781], [0,0,0,0], [9E9, 9E9, 9E9, 9E9, 9E9, 9E9]];
	VAR robtarget Openhole_3294 := [[449.06, -3, 181.35], [-0.053831, 0.705055, 0.705181, -0.052147], [0,0,0,0], [9E9, 9E9, 9E9, 9E9, 9E9, 9E9]];
	VAR robtarget Openhole_3295 := [[448.57, -3, 181.42], [-0.055497, 0.704926, 0.705304, -0.050458], [0,0,0,0], [9E9, 9E9, 9E9, 9E9, 9E9, 9E9]];
	VAR robtarget Openhole_3296 := [[448.07, -3.04, 181.5], [-0.05704, 0.704802, 0.705431, -0.048656], [0,0,0,0], [9E9, 9E9, 9E9, 9E9, 9E9, 9E9]];
	VAR robtarget Openhole_3297 := [[447.58, -3.09, 181.57], [-0.058549, 0.704679, 0.705555, -0.046825], [0,0,0,0], [9E9, 9E9, 9E9, 9E9, 9E9, 9E9]];
	VAR robtarget Openhole_3298 := [[447.09, -3.15, 181.65], [-0.059993, 0.704557, 0.705677, -0.044941], [0,0,0,0], [9E9, 9E9, 9E9, 9E9, 9E9, 9E9]];
	VAR robtarget Openhole_3299 := [[446.11, -3.31, 181.79], [-0.06277, 0.704315, 0.705912, -0.041089], [0,0,0,0], [9E9, 9E9, 9E9, 9E9, 9E9, 9E9]];
	VAR robtarget Openhole_3300 := [[437.9, -5.24, 182.82], [-0.08377, 0.702127, 0.707076, -0.006634], [0,0,0,0], [9E9, 9E9, 9E9, 9E9, 9E9, 9E9]];
	VAR robtarget Openhole_3301 := [[431.53, -6.32, 183.48], [-0.10098, 0.699859, 0.706863, 0.018548], [0,0,0,0], [9E9, 9E9, 9E9, 9E9, 9E9, 9E9]];
	VAR robtarget Openhole_3302 := [[423.12, -7.3, 184.26], [-0.124253, 0.696104, 0.705359, 0.049681], [0,0,0,0], [9E9, 9E9, 9E9, 9E9, 9E9, 9E9]];
	VAR robtarget Openhole_3303 := [[413.19, -8.06, 185.12], [-0.151403, 0.690708, 0.702118, 0.083849], [0,0,0,0], [9E9, 9E9, 9E9, 9E9, 9E9, 9E9]];
	VAR robtarget Openhole_3304 := [[394.36, -9.02, 186.6], [-0.198627, 0.678636, 0.692759, 0.141724], [0,0,0,0], [9E9, 9E9, 9E9, 9E9, 9E9, 9E9]];
	VAR robtarget Openhole_3305 := [[389.36, -9.02, 187.08], [-0.210565, 0.675028, 0.689909, 0.155004], [0,0,0,0], [9E9, 9E9, 9E9, 9E9, 9E9, 9E9]];
	VAR robtarget Openhole_3306 := [[362.36, -9.02, 187.16], [-0.183051, 0.683002, 0.683002, 0.183051], [0,0,0,0], [9E9, 9E9, 9E9, 9E9, 9E9, 9E9]];
	VAR robtarget Openhole_3307 := [[362.36, -10.02, 186.59], [-0.183051, 0.683002, 0.683002, 0.183051], [0,0,0,0], [9E9, 9E9, 9E9, 9E9, 9E9, 9E9]];
	VAR robtarget Openhole_3308 := [[389.36, -10.02, 186.5], [-0.207765, 0.675895, 0.68926, 0.157862], [0,0,0,0], [9E9, 9E9, 9E9, 9E9, 9E9, 9E9]];
	VAR robtarget Openhole_3309 := [[394.36, -10.02, 186.07], [-0.195755, 0.67947, 0.692153, 0.144652], [0,0,0,0], [9E9, 9E9, 9E9, 9E9, 9E9, 9E9]];
	VAR robtarget Openhole_3310 := [[406.83, -9.43, 185.23], [-0.165039, 0.687577, 0.698887, 0.107502], [0,0,0,0], [9E9, 9E9, 9E9, 9E9, 9E9, 9E9]];
	VAR robtarget Openhole_3311 := [[420.77, -8.72, 184.14], [-0.126894, 0.695628, 0.704388, 0.061949], [0,0,0,0], [9E9, 9E9, 9E9, 9E9, 9E9, 9E9]];
	VAR robtarget Openhole_3312 := [[431.69, -7.82, 183.21], [-0.095561, 0.70062, 0.706734, 0.022953], [0,0,0,0], [9E9, 9E9, 9E9, 9E9, 9E9, 9E9]];
	VAR robtarget Openhole_3313 := [[439.1, -6.9, 182.5], [-0.074331, 0.703189, 0.707088, -0.005184], [0,0,0,0], [9E9, 9E9, 9E9, 9E9, 9E9, 9E9]];
	VAR robtarget Openhole_3314 := [[445.46, -5.78, 181.8], [-0.056758, 0.704825, 0.706443, -0.030633], [0,0,0,0], [9E9, 9E9, 9E9, 9E9, 9E9, 9E9]];
	VAR robtarget Openhole_3315 := [[446.45, -5.65, 181.68], [-0.053854, 0.705053, 0.706269, -0.034411], [0,0,0,0], [9E9, 9E9, 9E9, 9E9, 9E9, 9E9]];
	VAR robtarget Openhole_3316 := [[446.94, -5.6, 181.61], [-0.052346, 0.705167, 0.706177, -0.036256], [0,0,0,0], [9E9, 9E9, 9E9, 9E9, 9E9, 9E9]];
	VAR robtarget Openhole_3317 := [[447.43, -5.56, 181.55], [-0.050795, 0.70528, 0.706082, -0.038063], [0,0,0,0], [9E9, 9E9, 9E9, 9E9, 9E9, 9E9]];
	VAR robtarget Openhole_3318 := [[447.93, -5.54, 181.49], [-0.049188, 0.705394, 0.705985, -0.039823], [0,0,0,0], [9E9, 9E9, 9E9, 9E9, 9E9, 9E9]];
	VAR robtarget Openhole_3319 := [[448.42, -5.54, 181.42], [-0.047517, 0.705508, 0.705887, -0.04152], [0,0,0,0], [9E9, 9E9, 9E9, 9E9, 9E9, 9E9]];
	VAR robtarget Openhole_3320 := [[448.92, -5.55, 181.36], [-0.045805, 0.705622, 0.705787, -0.043176], [0,0,0,0], [9E9, 9E9, 9E9, 9E9, 9E9, 9E9]];
	VAR robtarget Openhole_3321 := [[450.41, -5.64, 181.16], [-0.040461, 0.705948, 0.705481, -0.047924], [0,0,0,0], [9E9, 9E9, 9E9, 9E9, 9E9, 9E9]];
	VAR robtarget Openhole_3322 := [[456.83, -6.26, 180.38], [-0.01646, 0.706915, 0.703881, -0.06747], [0,0,0,0], [9E9, 9E9, 9E9, 9E9, 9E9, 9E9]];
	VAR robtarget Openhole_3323 := [[457.32, -6.28, 180.32], [-0.014684, 0.706954, 0.703728, -0.069044], [0,0,0,0], [9E9, 9E9, 9E9, 9E9, 9E9, 9E9]];
	VAR robtarget Openhole_3324 := [[457.82, -6.3, 180.26], [-0.012942, 0.706988, 0.703568, -0.07065], [0,0,0,0], [9E9, 9E9, 9E9, 9E9, 9E9, 9E9]];
	VAR robtarget Openhole_3325 := [[458.32, -6.3, 180.2], [-0.011242, 0.707017, 0.703401, -0.072297], [0,0,0,0], [9E9, 9E9, 9E9, 9E9, 9E9, 9E9]];
	VAR robtarget Openhole_3326 := [[458.81, -6.29, 180.14], [-0.009573, 0.707042, 0.703227, -0.073969], [0,0,0,0], [9E9, 9E9, 9E9, 9E9, 9E9, 9E9]];
	VAR robtarget Openhole_3327 := [[459.31, -6.28, 180.08], [-0.007909, 0.707063, 0.703049, -0.075645], [0,0,0,0], [9E9, 9E9, 9E9, 9E9, 9E9, 9E9]];
	VAR robtarget Openhole_3328 := [[460.3, -6.24, 179.95], [-0.00467, 0.707091, 0.702673, -0.079065], [0,0,0,0], [9E9, 9E9, 9E9, 9E9, 9E9, 9E9]];
	VAR robtarget Openhole_3329 := [[461.29, -6.17, 179.82], [-0.00153, 0.707105, 0.702271, -0.082554], [0,0,0,0], [9E9, 9E9, 9E9, 9E9, 9E9, 9E9]];
	VAR robtarget Openhole_3330 := [[463.75, -5.92, 179.48], [0.005999, 0.707081, 0.701167, -0.091463], [0,0,0,0], [9E9, 9E9, 9E9, 9E9, 9E9, 9E9]];
	VAR robtarget Openhole_3331 := [[472.09, -4.91, 178.21], [0.030746, 0.706438, 0.696614, -0.121361], [0,0,0,0], [9E9, 9E9, 9E9, 9E9, 9E9, 9E9]];
	VAR robtarget Openhole_3332 := [[477.03, -4.63, 177.46], [0.04616, 0.705599, 0.693635, -0.137372], [0,0,0,0], [9E9, 9E9, 9E9, 9E9, 9E9, 9E9]];
	VAR robtarget Openhole_3333 := [[478.51, -4.61, 177.25], [0.050952, 0.705269, 0.692726, -0.141882], [0,0,0,0], [9E9, 9E9, 9E9, 9E9, 9E9, 9E9]];
	VAR robtarget Openhole_3334 := [[479.01, -4.61, 177.18], [0.052565, 0.70515, 0.692423, -0.143354], [0,0,0,0], [9E9, 9E9, 9E9, 9E9, 9E9, 9E9]];
	VAR robtarget Openhole_3335 := [[484.46, -4.79, 176.49], [0.070627, 0.703571, 0.689073, -0.158676], [0,0,0,0], [9E9, 9E9, 9E9, 9E9, 9E9, 9E9]];
	VAR robtarget Openhole_3336 := [[491.4, -5.38, 175.78], [0.093965, 0.700836, 0.684814, -0.176153], [0,0,0,0], [9E9, 9E9, 9E9, 9E9, 9E9, 9E9]];
	VAR robtarget Openhole_3337 := [[500.82, -6.37, 175.03], [0.124537, 0.696054, 0.678909, -0.197692], [0,0,0,0], [9E9, 9E9, 9E9, 9E9, 9E9, 9E9]];
	VAR robtarget Openhole_3338 := [[503.8, -6.51, 174.74], [0.133273, 0.694434, 0.676855, -0.204615], [0,0,0,0], [9E9, 9E9, 9E9, 9E9, 9E9, 9E9]];
	VAR robtarget Openhole_3339 := [[504.3, -6.51, 174.68], [0.134642, 0.69417, 0.676492, -0.205812], [0,0,0,0], [9E9, 9E9, 9E9, 9E9, 9E9, 9E9]];
	VAR robtarget Openhole_3340 := [[504.33, -6.51, 174.67], [0.134728, 0.694153, 0.676471, -0.20588], [0,0,0,0], [9E9, 9E9, 9E9, 9E9, 9E9, 9E9]];
	VAR robtarget Openhole_3341 := [[509.32, -6.51, 174.07], [0.183051, 0.683002, 0.683002, -0.183051], [0,0,0,0], [9E9, 9E9, 9E9, 9E9, 9E9, 9E9]];
	VAR robtarget Openhole_3342 := [[536.32, -6.51, 173.99], [0.183051, 0.683002, 0.683002, -0.183051], [0,0,0,0], [9E9, 9E9, 9E9, 9E9, 9E9, 9E9]];
	VAR robtarget Openhole_3343 := [[536.33, -7.39, 174.5], [0.183051, 0.683002, 0.683002, -0.183051], [0,0,0,0], [9E9, 9E9, 9E9, 9E9, 9E9, 9E9]];
	VAR robtarget Openhole_3344 := [[509.33, -7.39, 174.58], [0.183051, 0.683002, 0.683002, -0.183051], [0,0,0,0], [9E9, 9E9, 9E9, 9E9, 9E9, 9E9]];
	VAR robtarget Openhole_3345 := [[504.33, -7.39, 175.14], [0.13731, 0.693647, 0.677232, -0.203365], [0,0,0,0], [9E9, 9E9, 9E9, 9E9, 9E9, 9E9]];
	VAR robtarget Openhole_3346 := [[503.78, -7.39, 175.2], [0.135804, 0.693943, 0.677623, -0.202055], [0,0,0,0], [9E9, 9E9, 9E9, 9E9, 9E9, 9E9]];
	VAR robtarget Openhole_3347 := [[499.31, -7.22, 175.62], [0.122805, 0.696361, 0.68071, -0.191399], [0,0,0,0], [9E9, 9E9, 9E9, 9E9, 9E9, 9E9]];
	VAR robtarget Openhole_3348 := [[487.39, -6.24, 176.62], [0.084352, 0.702058, 0.688184, -0.162491], [0,0,0,0], [9E9, 9E9, 9E9, 9E9, 9E9, 9E9]];
	VAR robtarget Openhole_3349 := [[481.43, -5.99, 177.27], [0.064779, 0.704133, 0.691832, -0.146181], [0,0,0,0], [9E9, 9E9, 9E9, 9E9, 9E9, 9E9]];
	VAR robtarget Openhole_3350 := [[479.94, -5.98, 177.46], [0.059969, 0.704559, 0.69274, -0.141815], [0,0,0,0], [9E9, 9E9, 9E9, 9E9, 9E9, 9E9]];
	VAR robtarget Openhole_3351 := [[479.45, -5.98, 177.52], [0.058381, 0.704693, 0.693042, -0.140331], [0,0,0,0], [9E9, 9E9, 9E9, 9E9, 9E9, 9E9]];
	VAR robtarget Openhole_3352 := [[474.99, -6.17, 178.13], [0.044461, 0.705708, 0.695742, -0.126265], [0,0,0,0], [9E9, 9E9, 9E9, 9E9, 9E9, 9E9]];
	VAR robtarget Openhole_3353 := [[470.08, -6.73, 178.85], [0.030016, 0.706469, 0.698637, -0.109115], [0,0,0,0], [9E9, 9E9, 9E9, 9E9, 9E9, 9E9]];
	VAR robtarget Openhole_3354 := [[463.75, -7.88, 179.76], [0.012505, 0.706996, 0.701983, -0.084971], [0,0,0,0], [9E9, 9E9, 9E9, 9E9, 9E9, 9E9]];
	VAR robtarget Openhole_3355 := [[456.91, -9.15, 180.58], [-0.006457, 0.707077, 0.704717, -0.05809], [0,0,0,0], [9E9, 9E9, 9E9, 9E9, 9E9, 9E9]];
	VAR robtarget Openhole_3356 := [[453.96, -9.56, 180.88], [-0.015183, 0.706944, 0.705557, -0.046786], [0,0,0,0], [9E9, 9E9, 9E9, 9E9, 9E9, 9E9]];
	VAR robtarget Openhole_3357 := [[453.46, -9.61, 180.93], [-0.016674, 0.70691, 0.705678, -0.044922], [0,0,0,0], [9E9, 9E9, 9E9, 9E9, 9E9, 9E9]];
	VAR robtarget Openhole_3358 := [[452.96, -9.66, 180.98], [-0.018209, 0.706872, 0.705793, -0.043091], [0,0,0,0], [9E9, 9E9, 9E9, 9E9, 9E9, 9E9]];
	VAR robtarget Openhole_3359 := [[451.47, -9.76, 181.11], [-0.022962, 0.706734, 0.7061, -0.037717], [0,0,0,0], [9E9, 9E9, 9E9, 9E9, 9E9, 9E9]];
	VAR robtarget Openhole_3360 := [[450.48, -9.77, 181.2], [-0.026313, 0.706617, 0.706275, -0.034296], [0,0,0,0], [9E9, 9E9, 9E9, 9E9, 9E9, 9E9]];
	VAR robtarget Openhole_3361 := [[447, -9.62, 181.51], [-0.038666, 0.706049, 0.706734, -0.022968], [0,0,0,0], [9E9, 9E9, 9E9, 9E9, 9E9, 9E9]];
	VAR robtarget Openhole_3362 := [[445.01, -9.52, 181.7], [-0.045742, 0.705626, 0.706913, -0.016534], [0,0,0,0], [9E9, 9E9, 9E9, 9E9, 9E9, 9E9]];
	VAR robtarget Openhole_3363 := [[443.51, -9.49, 181.84], [-0.050858, 0.705275, 0.707013, -0.011518], [0,0,0,0], [9E9, 9E9, 9E9, 9E9, 9E9, 9E9]];
	VAR robtarget Openhole_3364 := [[433.06, -9.93, 182.73], [-0.084108, 0.702087, 0.706651, 0.025374], [0,0,0,0], [9E9, 9E9, 9E9, 9E9, 9E9, 9E9]];
	VAR robtarget Openhole_3365 := [[412.13, -10.76, 184.26], [-0.146006, 0.691869, 0.700611, 0.095627], [0,0,0,0], [9E9, 9E9, 9E9, 9E9, 9E9, 9E9]];
	VAR robtarget Openhole_3366 := [[397.17, -11.31, 185.18], [-0.184985, 0.682481, 0.692951, 0.14078], [0,0,0,0], [9E9, 9E9, 9E9, 9E9, 9E9, 9E9]];
	VAR robtarget Openhole_3367 := [[394.36, -11.45, 185.31], [-0.191641, 0.680642, 0.691266, 0.148835], [0,0,0,0], [9E9, 9E9, 9E9, 9E9, 9E9, 9E9]];
	VAR robtarget Openhole_3368 := [[389.36, -11.45, 185.68], [-0.203756, 0.677114, 0.688312, 0.161945], [0,0,0,0], [9E9, 9E9, 9E9, 9E9, 9E9, 9E9]];
	VAR robtarget Openhole_3369 := [[360.28, -11.45, 185.77], [-0.183051, 0.683002, 0.683002, 0.183051], [0,0,0,0], [9E9, 9E9, 9E9, 9E9, 9E9, 9E9]];
	VAR robtarget Openhole_3370 := [[360.24, -35.51, 171.87], [-0.183051, 0.683002, 0.683002, 0.183051], [0,0,0,0], [9E9, 9E9, 9E9, 9E9, 9E9, 9E9]];
	VAR robtarget Openhole_3371 := [[389.32, -35.51, 171.78], [-0.135275, 0.694047, 0.668747, 0.229734], [0,0,0,0], [9E9, 9E9, 9E9, 9E9, 9E9, 9E9]];
	VAR robtarget Openhole_3372 := [[394.32, -35.51, 172.58], [-0.121448, 0.696599, 0.672551, 0.218346], [0,0,0,0], [9E9, 9E9, 9E9, 9E9, 9E9, 9E9]];
	VAR robtarget Openhole_3373 := [[394.71, -35.54, 172.62], [-0.120254, 0.696806, 0.672827, 0.217495], [0,0,0,0], [9E9, 9E9, 9E9, 9E9, 9E9, 9E9]];
	VAR robtarget Openhole_3374 := [[395.19, -35.69, 172.62], [-0.118454, 0.697114, 0.673047, 0.216814], [0,0,0,0], [9E9, 9E9, 9E9, 9E9, 9E9, 9E9]];
	VAR robtarget Openhole_3375 := [[399.53, -36.88, 172.74], [-0.102399, 0.699653, 0.675269, 0.20979], [0,0,0,0], [9E9, 9E9, 9E9, 9E9, 9E9, 9E9]];
	VAR robtarget Openhole_3376 := [[404.89, -38.02, 173.18], [-0.082868, 0.702234, 0.678331, 0.199666], [0,0,0,0], [9E9, 9E9, 9E9, 9E9, 9E9, 9E9]];
	VAR robtarget Openhole_3377 := [[408.32, -38.6, 173.58], [-0.070465, 0.703587, 0.680407, 0.192474], [0,0,0,0], [9E9, 9E9, 9E9, 9E9, 9E9, 9E9]];
	VAR robtarget Openhole_3378 := [[408.81, -38.7, 173.63], [-0.068623, 0.703769, 0.680692, 0.191463], [0,0,0,0], [9E9, 9E9, 9E9, 9E9, 9E9, 9E9]];
	VAR robtarget Openhole_3379 := [[419.27, -38.7, 175.61], [-0.034833, 0.706248, 0.688189, 0.162468], [0,0,0,0], [9E9, 9E9, 9E9, 9E9, 9E9, 9E9]];
	VAR robtarget Openhole_3380 := [[418.78, -38.66, 175.53], [-0.036595, 0.706159, 0.687883, 0.163758], [0,0,0,0], [9E9, 9E9, 9E9, 9E9, 9E9, 9E9]];
	VAR robtarget Openhole_3381 := [[412.88, -38.13, 174.6], [-0.057443, 0.70477, 0.684131, 0.178788], [0,0,0,0], [9E9, 9E9, 9E9, 9E9, 9E9, 9E9]];
	VAR robtarget Openhole_3382 := [[406.49, -37.23, 173.8], [-0.080337, 0.702528, 0.680202, 0.193197], [0,0,0,0], [9E9, 9E9, 9E9, 9E9, 9E9, 9E9]];
	VAR robtarget Openhole_3383 := [[401.11, -36.21, 173.33], [-0.099719, 0.70004, 0.677055, 0.203951], [0,0,0,0], [9E9, 9E9, 9E9, 9E9, 9E9, 9E9]];
	VAR robtarget Openhole_3384 := [[395.29, -34.79, 173.1], [-0.120814, 0.696709, 0.673931, 0.214049], [0,0,0,0], [9E9, 9E9, 9E9, 9E9, 9E9, 9E9]];
	VAR robtarget Openhole_3385 := [[394.23, -34.53, 173.08], [-0.124548, 0.696052, 0.673379, 0.215779], [0,0,0,0], [9E9, 9E9, 9E9, 9E9, 9E9, 9E9]];
	VAR robtarget Openhole_3386 := [[389.32, -34.53, 172.35], [-0.138067, 0.693497, 0.669666, 0.22704], [0,0,0,0], [9E9, 9E9, 9E9, 9E9, 9E9, 9E9]];
	VAR robtarget Openhole_3387 := [[362.32, -34.53, 172.43], [-0.183051, 0.683002, 0.683002, 0.183051], [0,0,0,0], [9E9, 9E9, 9E9, 9E9, 9E9, 9E9]];
	VAR robtarget Openhole_3388 := [[362.32, -33.65, 172.94], [-0.183051, 0.683002, 0.683002, 0.183051], [0,0,0,0], [9E9, 9E9, 9E9, 9E9, 9E9, 9E9]];
	VAR robtarget Openhole_3389 := [[389.32, -33.65, 172.85], [-0.140548, 0.692998, 0.670475, 0.224641], [0,0,0,0], [9E9, 9E9, 9E9, 9E9, 9E9, 9E9]];
	VAR robtarget Openhole_3390 := [[394.32, -33.65, 173.56], [-0.126846, 0.695636, 0.674224, 0.213123], [0,0,0,0], [9E9, 9E9, 9E9, 9E9, 9E9, 9E9]];
	VAR robtarget Openhole_3391 := [[395, -33.77, 173.59], [-0.124628, 0.696037, 0.674629, 0.211838], [0,0,0,0], [9E9, 9E9, 9E9, 9E9, 9E9, 9E9]];
	VAR robtarget Openhole_3392 := [[402.33, -35.28, 173.95], [-0.098861, 0.700162, 0.678763, 0.198195], [0,0,0,0], [9E9, 9E9, 9E9, 9E9, 9E9, 9E9]];
	VAR robtarget Openhole_3393 := [[408.72, -36.33, 174.54], [-0.076193, 0.70299, 0.682573, 0.184645], [0,0,0,0], [9E9, 9E9, 9E9, 9E9, 9E9, 9E9]];
	VAR robtarget Openhole_3394 := [[414.63, -37, 175.3], [-0.055342, 0.704938, 0.686246, 0.170488], [0,0,0,0], [9E9, 9E9, 9E9, 9E9, 9E9, 9E9]];
	VAR robtarget Openhole_3395 := [[420.55, -37.36, 176.22], [-0.03488, 0.706246, 0.689998, 0.154604], [0,0,0,0], [9E9, 9E9, 9E9, 9E9, 9E9, 9E9]];
	VAR robtarget Openhole_3396 := [[424, -37.4, 176.82], [-0.023254, 0.706724, 0.692184, 0.144504], [0,0,0,0], [9E9, 9E9, 9E9, 9E9, 9E9, 9E9]];
	VAR robtarget Openhole_3397 := [[424.49, -37.4, 176.91], [-0.021619, 0.706776, 0.692495, 0.143005], [0,0,0,0], [9E9, 9E9, 9E9, 9E9, 9E9, 9E9]];
	VAR robtarget Openhole_3398 := [[431.37, -37.13, 178.17], [0.000765, 0.707106, 0.696694, 0.120904], [0,0,0,0], [9E9, 9E9, 9E9, 9E9, 9E9, 9E9]];
	VAR robtarget Openhole_3399 := [[437.27, -36.86, 179.23], [0.020047, 0.706823, 0.699837, 0.101136], [0,0,0,0], [9E9, 9E9, 9E9, 9E9, 9E9, 9E9]];
	VAR robtarget Openhole_3400 := [[437.76, -36.86, 179.31], [0.021731, 0.706773, 0.700067, 0.099527], [0,0,0,0], [9E9, 9E9, 9E9, 9E9, 9E9, 9E9]];
	VAR robtarget Openhole_3401 := [[438.25, -36.86, 179.4], [0.023419, 0.706719, 0.700294, 0.097919], [0,0,0,0], [9E9, 9E9, 9E9, 9E9, 9E9, 9E9]];
	VAR robtarget Openhole_3402 := [[442.19, -37.1, 180.06], [0.037673, 0.706102, 0.701892, 0.085717], [0,0,0,0], [9E9, 9E9, 9E9, 9E9, 9E9, 9E9]];
	VAR robtarget Openhole_3403 := [[443.17, -37.22, 180.22], [0.04143, 0.705892, 0.702234, 0.082867], [0,0,0,0], [9E9, 9E9, 9E9, 9E9, 9E9, 9E9]];
	VAR robtarget Openhole_3404 := [[444.14, -37.38, 180.38], [0.045289, 0.705655, 0.70255, 0.080149], [0,0,0,0], [9E9, 9E9, 9E9, 9E9, 9E9, 9E9]];
	VAR robtarget Openhole_3405 := [[445.11, -37.59, 180.54], [0.049261, 0.705389, 0.702836, 0.077594], [0,0,0,0], [9E9, 9E9, 9E9, 9E9, 9E9, 9E9]];
	VAR robtarget Openhole_3406 := [[446.06, -37.84, 180.71], [0.053344, 0.705092, 0.703095, 0.07522], [0,0,0,0], [9E9, 9E9, 9E9, 9E9, 9E9, 9E9]];
	VAR robtarget Openhole_3407 := [[447.02, -38.07, 180.88], [0.057349, 0.704777, 0.703357, 0.072728], [0,0,0,0], [9E9, 9E9, 9E9, 9E9, 9E9, 9E9]];
	VAR robtarget Openhole_3408 := [[447.51, -38.14, 180.96], [0.059258, 0.704619, 0.703498, 0.071347], [0,0,0,0], [9E9, 9E9, 9E9, 9E9, 9E9, 9E9]];
	VAR robtarget Openhole_3409 := [[448, -38.2, 181.05], [0.061117, 0.704461, 0.703643, 0.069899], [0,0,0,0], [9E9, 9E9, 9E9, 9E9, 9E9, 9E9]];
	VAR robtarget Openhole_3410 := [[448.49, -38.23, 181.14], [0.062863, 0.704307, 0.703799, 0.06832], [0,0,0,0], [9E9, 9E9, 9E9, 9E9, 9E9, 9E9]];
	VAR robtarget Openhole_3411 := [[448.98, -38.23, 181.23], [0.064536, 0.704156, 0.703958, 0.066662], [0,0,0,0], [9E9, 9E9, 9E9, 9E9, 9E9, 9E9]];
	VAR robtarget Openhole_3412 := [[449.47, -38.19, 181.32], [0.066052, 0.704015, 0.704126, 0.064859], [0,0,0,0], [9E9, 9E9, 9E9, 9E9, 9E9, 9E9]];
	VAR robtarget Openhole_3413 := [[449.96, -38.12, 181.41], [0.067484, 0.703879, 0.704295, 0.062992], [0,0,0,0], [9E9, 9E9, 9E9, 9E9, 9E9, 9E9]];
	VAR robtarget Openhole_3414 := [[450.91, -37.89, 181.59], [0.069981, 0.703635, 0.704641, 0.058997], [0,0,0,0], [9E9, 9E9, 9E9, 9E9, 9E9, 9E9]];
	VAR robtarget Openhole_3415 := [[459, -35.6, 182.84], [0.089464, 0.701424, 0.706704, 0.023849], [0,0,0,0], [9E9, 9E9, 9E9, 9E9, 9E9, 9E9]];
	VAR robtarget Openhole_3416 := [[464.29, -34.25, 183.49], [0.102303, 0.699667, 0.707106, 0.001331], [0,0,0,0], [9E9, 9E9, 9E9, 9E9, 9E9, 9E9]];
	VAR robtarget Openhole_3417 := [[471.13, -32.95, 184.22], [0.119807, 0.696883, 0.706627, -0.026037], [0,0,0,0], [9E9, 9E9, 9E9, 9E9, 9E9, 9E9]];
	VAR robtarget Openhole_3418 := [[479.02, -31.9, 184.98], [0.140498, 0.693008, 0.704925, -0.055507], [0,0,0,0], [9E9, 9E9, 9E9, 9E9, 9E9, 9E9]];
	VAR robtarget Openhole_3419 := [[488.95, -31.06, 185.89], [0.166342, 0.687263, 0.701411, -0.089567], [0,0,0,0], [9E9, 9E9, 9E9, 9E9, 9E9, 9E9]];
	VAR robtarget Openhole_3420 := [[504.38, -30.16, 187.2], [0.203574, 0.677169, 0.69366, -0.137245], [0,0,0,0], [9E9, 9E9, 9E9, 9E9, 9E9, 9E9]];
	VAR robtarget Openhole_3421 := [[509.37, -30.16, 187.73], [0.183051, 0.683002, 0.683002, -0.183051], [0,0,0,0], [9E9, 9E9, 9E9, 9E9, 9E9, 9E9]];
	VAR robtarget Openhole_3422 := [[536.37, -30.16, 187.65], [0.183051, 0.683002, 0.683002, -0.183051], [0,0,0,0], [9E9, 9E9, 9E9, 9E9, 9E9, 9E9]];
	VAR robtarget Openhole_3423 := [[536.36, -29.28, 187.14], [0.183051, 0.683002, 0.683002, -0.183051], [0,0,0,0], [9E9, 9E9, 9E9, 9E9, 9E9, 9E9]];
	VAR robtarget Openhole_3424 := [[509.37, -29.28, 187.22], [0.183051, 0.683002, 0.683002, -0.183051], [0,0,0,0], [9E9, 9E9, 9E9, 9E9, 9E9, 9E9]];
	VAR robtarget Openhole_3425 := [[504.36, -29.28, 186.73], [0.201023, 0.677931, 0.693151, -0.139792], [0,0,0,0], [9E9, 9E9, 9E9, 9E9, 9E9, 9E9]];
	VAR robtarget Openhole_3426 := [[485.08, -30.34, 185.19], [0.153258, 0.690298, 0.702589, -0.079801], [0,0,0,0], [9E9, 9E9, 9E9, 9E9, 9E9, 9E9]];
	VAR robtarget Openhole_3427 := [[476.14, -31.11, 184.42], [0.129335, 0.695178, 0.705431, -0.048649], [0,0,0,0], [9E9, 9E9, 9E9, 9E9, 9E9, 9E9]];
	VAR robtarget Openhole_3428 := [[468.24, -32.14, 183.69], [0.10807, 0.6988, 0.706851, -0.019019], [0,0,0,0], [9E9, 9E9, 9E9, 9E9, 9E9, 9E9]];
	VAR robtarget Openhole_3429 := [[461.89, -33.32, 183.03], [0.091429, 0.701171, 0.707078, 0.006434], [0,0,0,0], [9E9, 9E9, 9E9, 9E9, 9E9, 9E9]];
	VAR robtarget Openhole_3430 := [[456.11, -34.79, 182.33], [0.07724, 0.702876, 0.706425, 0.031048], [0,0,0,0], [9E9, 9E9, 9E9, 9E9, 9E9, 9E9]];
	VAR robtarget Openhole_3431 := [[451.33, -36.06, 181.63], [0.065374, 0.704078, 0.705224, 0.051563], [0,0,0,0], [9E9, 9E9, 9E9, 9E9, 9E9, 9E9]];
	VAR robtarget Openhole_3432 := [[450.85, -36.17, 181.55], [0.064084, 0.704197, 0.705076, 0.053546], [0,0,0,0], [9E9, 9E9, 9E9, 9E9, 9E9, 9E9]];
	VAR robtarget Openhole_3433 := [[449.87, -36.33, 181.39], [0.06134, 0.704441, 0.704773, 0.057397], [0,0,0,0], [9E9, 9E9, 9E9, 9E9, 9E9, 9E9]];
	VAR robtarget Openhole_3434 := [[449.38, -36.38, 181.31], [0.059843, 0.70457, 0.704622, 0.059225], [0,0,0,0], [9E9, 9E9, 9E9, 9E9, 9E9, 9E9]];
	VAR robtarget Openhole_3435 := [[448.89, -36.4, 181.23], [0.058219, 0.704706, 0.704476, 0.060944], [0,0,0,0], [9E9, 9E9, 9E9, 9E9, 9E9, 9E9]];
	VAR robtarget Openhole_3436 := [[448.4, -36.38, 181.14], [0.056494, 0.704846, 0.704334, 0.062562], [0,0,0,0], [9E9, 9E9, 9E9, 9E9, 9E9, 9E9]];
	VAR robtarget Openhole_3437 := [[447.91, -36.33, 181.06], [0.054669, 0.70499, 0.704199, 0.064063], [0,0,0,0], [9E9, 9E9, 9E9, 9E9, 9E9, 9E9]];
	VAR robtarget Openhole_3438 := [[447.42, -36.26, 180.98], [0.052764, 0.705135, 0.70407, 0.065466], [0,0,0,0], [9E9, 9E9, 9E9, 9E9, 9E9, 9E9]];
	VAR robtarget Openhole_3439 := [[446.93, -36.18, 180.9], [0.050829, 0.705278, 0.703942, 0.066826], [0,0,0,0], [9E9, 9E9, 9E9, 9E9, 9E9, 9E9]];
	VAR robtarget Openhole_3440 := [[442.57, -35.3, 180.24], [0.033031, 0.706335, 0.70273, 0.078551], [0,0,0,0], [9E9, 9E9, 9E9, 9E9, 9E9, 9E9]];
	VAR robtarget Openhole_3441 := [[440.11, -35, 179.88], [0.023654, 0.706711, 0.701891, 0.085728], [0,0,0,0], [9E9, 9E9, 9E9, 9E9, 9E9, 9E9]];
	VAR robtarget Openhole_3442 := [[439.13, -34.94, 179.74], [0.020061, 0.706822, 0.701513, 0.088768], [0,0,0,0], [9E9, 9E9, 9E9, 9E9, 9E9, 9E9]];
	VAR robtarget Openhole_3443 := [[437.15, -34.9, 179.44], [0.013161, 0.706984, 0.700681, 0.095108], [0,0,0,0], [9E9, 9E9, 9E9, 9E9, 9E9, 9E9]];
	VAR robtarget Openhole_3444 := [[436.66, -34.9, 179.36], [0.011491, 0.707013, 0.700458, 0.096738], [0,0,0,0], [9E9, 9E9, 9E9, 9E9, 9E9, 9E9]];
	VAR robtarget Openhole_3445 := [[431.24, -35.21, 178.48], [-0.005941, 0.707082, 0.697666, 0.115161], [0,0,0,0], [9E9, 9E9, 9E9, 9E9, 9E9, 9E9]];
	VAR robtarget Openhole_3446 := [[424.35, -35.64, 177.31], [-0.02776, 0.706562, 0.693534, 0.137877], [0,0,0,0], [9E9, 9E9, 9E9, 9E9, 9E9, 9E9]];
	VAR robtarget Openhole_3447 := [[421.88, -35.68, 176.9], [-0.035834, 0.706198, 0.691992, 0.145419], [0,0,0,0], [9E9, 9E9, 9E9, 9E9, 9E9, 9E9]];
	VAR robtarget Openhole_3448 := [[421.39, -35.68, 176.82], [-0.037472, 0.706113, 0.691683, 0.146882], [0,0,0,0], [9E9, 9E9, 9E9, 9E9, 9E9, 9E9]];
	VAR robtarget Openhole_3449 := [[415.95, -35.48, 176.02], [-0.05586, 0.704897, 0.688275, 0.162103], [0,0,0,0], [9E9, 9E9, 9E9, 9E9, 9E9, 9E9]];
	VAR robtarget Openhole_3450 := [[410.02, -34.94, 175.28], [-0.076392, 0.702968, 0.684599, 0.176987], [0,0,0,0], [9E9, 9E9, 9E9, 9E9, 9E9, 9E9]];
	VAR robtarget Openhole_3451 := [[403.61, -34.06, 174.69], [-0.098744, 0.700178, 0.68073, 0.19133], [0,0,0,0], [9E9, 9E9, 9E9, 9E9, 9E9, 9E9]];
	VAR robtarget Openhole_3452 := [[395.25, -32.64, 174.22], [-0.127228, 0.695567, 0.675807, 0.208051], [0,0,0,0], [9E9, 9E9, 9E9, 9E9, 9E9, 9E9]];
	VAR robtarget Openhole_3453 := [[394.32, -32.55, 174.14], [-0.130064, 0.695042, 0.675204, 0.21], [0,0,0,0], [9E9, 9E9, 9E9, 9E9, 9E9, 9E9]];
	VAR robtarget Openhole_3454 := [[389.32, -32.55, 173.49], [-0.143691, 0.692353, 0.671487, 0.221596], [0,0,0,0], [9E9, 9E9, 9E9, 9E9, 9E9, 9E9]];
